KUKA KRL program: EPS_2_251806_MH43A_A_20260212042237.src

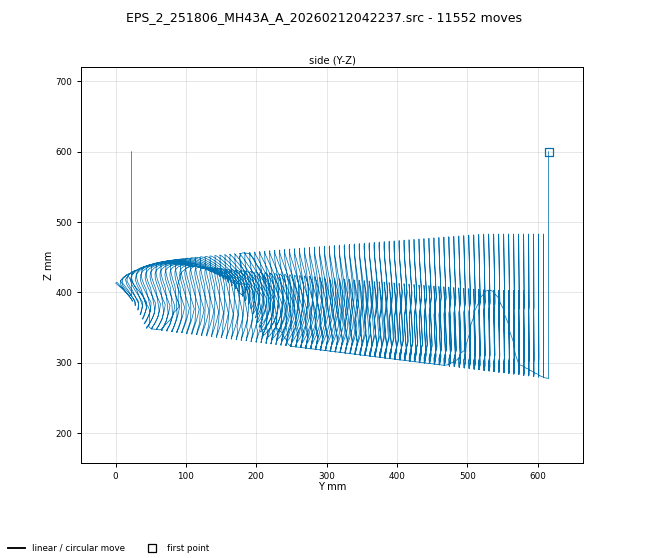
[picture p0: tool path of EPS_2_251806_MH43A_A_20260212042237.src, 11552 of 11554 moves have a stored position in this frame; points joined in program order, loops and branches not executed]
&ACCESS RVP
&REL 4
&COMMENT QRS 19112012
&PARAM EDITMASK = *
DEF PART()
EXT BAS (BAS_COMMAND :IN,REAL :IN )
INT I
BAS (#INITMOV,0 )

;KUKA QRS Post kuka4.cps  Date:22-06-2017 !

File_ID=3015

QRS_PRE_INIT()

;Init var - Until changes are made in qrs_pre_init
Outlet_Square_prg=0
Inlet_1_Square_prg=0
Inlet_2_Square_prg=0
Inlet_3_Square_prg=0
Inlet_4_Square_prg=0
Inlet_5_Square_prg=0

Outlet_1={X 0.000, Y 526.370, Z 382.500, B 0.000, E1 0.000 }
Inlet_1={X 0.000, Y 532.170, Z 302.500, B 0.000, E1 128.000 }
Outlet_1_type=201
Inlet_1_type=201
;QRS#1=Sidecore dimensions
;QRS#2=200-8" PVC SDR 35
;QRS#3=200-8" PVC SDR 35
;QRS#4=
;QRS#5=
;QRS#6=
;QRS#7=
;QRS#8=
;QRS#9=12-08 PSX
;QRS#10=12-08 PSX
;QRS#11=
;QRS#12=
;QRS#13=
;QRS#14=
;QRS#15=
;QRS#16=1220x127x762 2,5'
;QRS#17=EPS Height
;QRS#18=483
;QRS#19=*
;QRS#20= UPDATED VERSION 22-06-2017
;QRS#21=*
Outlet_Square=0100
Inlet_1_Square=0100
Inlet_2_Square=0
Inlet_3_Square=0
Inlet_4_Square=0
Inlet_5_Square=0
Mill_Square=1
Outlet_Square_Prg=204
Inlet_1_Square_prg=204

QRS_INIT()

$ADVANCE=5

; T1
PTP {E1 173.621,E2 173.621}
PTP {X 0,Y 615.489,A -85,B 0,C 180,E1 173.621,E2 173.621,E3 0,E4 0,E5 0,E6 0}
QRS_SPEED_INIT()
LIN {X 0,Y 615.489,Z 600,A -85,B 0,C 180,E1 173.621,E2 173.621,E3 0,E4 0,E5 0,E6 0} C_VEL
LIN {X 0,Y 615.489,Z 287.877,A -85,B 0,C 180,E1 173.621,E2 173.621} C_VEL
LIN {X 0,Y 615.489,Z 279.7,A -85,B 0,C 180,E1 173.621,E2 173.621} C_VEL
LIN {X 0,Y 615.478,Z 277.7,A -85,B 0,C 180,E1 173.435,E2 173.435} C_VEL
LIN {X 0,Y 615.494,Z 277.879,A -85,B 0,C 180,E1 170.801,E2 170.801} C_VEL
LIN {X 0,Y 615.483,Z 281.025,A -85,B 0,C 180,E1 168.139,E2 168.139} C_VEL
LIN {X 0,Y 615.467,Z 284.295,A -85,B 0,C 180,E1 165.451,E2 165.451} C_VEL
LIN {X 0,Y 615.488,Z 287.642,A -85,B 0,C 180,E1 162.73,E2 162.73} C_VEL
LIN {X 0,Y 615.467,Z 291.126,A -85,B 0,C 180,E1 159.967,E2 159.967} C_VEL
LIN {X 0,Y 615.473,Z 294.079,A -85,B 0,C 180,E1 157.659,E2 157.659} C_VEL
LIN {X 0,Y 615.485,Z 297.487,A -85,B 0,C 180,E1 155.008,E2 155.008} C_VEL
LIN {X 0,Y 615.484,Z 299.412,A -85,B 0,C 180,E1 153.537,E2 153.537} C_VEL
LIN {X 0,Y 615.487,Z 313.298,A -85,B 0,C 180,E1 153.219,E2 153.219} C_VEL
LIN {X 0,Y 615.486,Z 325.134,A -85,B 0,C 180,E1 152.823,E2 152.823} C_VEL
LIN {X 0,Y 615.476,Z 337.354,A -85,B 0,C 180,E1 152.269,E2 152.269} C_VEL
LIN {X 0,Y 615.49,Z 348.526,A -85,B 0,C 180,E1 151.617,E2 151.617} C_VEL
LIN {X 0,Y 615.5,Z 358.718,A -85,B 0,C 180,E1 150.876,E2 150.876} C_VEL
LIN {X 0,Y 615.498,Z 368.21,A -85,B 0,C 180,E1 150.023,E2 150.023} C_VEL
LIN {X 0,Y 615.497,Z 376.7,A -85,B 0,C 180,E1 149.081,E2 149.081} C_VEL
LIN {X 0,Y 615.498,Z 383.506,A -85,B 0,C 180,E1 148.154,E2 148.154} C_VEL
LIN {X 0,Y 615.495,Z 389.434,A -85,B 0,C 180,E1 147.154,E2 147.154} C_VEL
LIN {X 0,Y 615.495,Z 394.786,A -85,B 0,C 180,E1 145.979,E2 145.979} C_VEL
LIN {X 0,Y 615.497,Z 398.663,A -85,B 0,C 180,E1 144.786,E2 144.786} C_VEL
LIN {X 0,Y 615.494,Z 401.179,A -85,B 0,C 180,E1 143.576,E2 143.576} C_VEL
LIN {X 0,Y 615.496,Z 402.068,A -85,B 0,C 180,E1 142.758,E2 142.758} C_VEL
LIN {X 0,Y 615.494,Z 402.388,A -85,B 0,C 180,E1 141.932,E2 141.932} C_VEL
LIN {X 0,Y 615.495,Z 401.915,A -85,B 0,C 180,E1 140.938,E2 140.938} C_VEL
LIN {X 0,Y 615.496,Z 400.472,A -85,B 0,C 180,E1 139.911,E2 139.911} C_VEL
LIN {X 0,Y 615.494,Z 398.079,A -85,B 0,C 180,E1 138.905,E2 138.905} C_VEL
LIN {X 0,Y 615.497,Z 394.741,A -85,B 0,C 180,E1 137.92,E2 137.92} C_VEL
LIN {X 0,Y 615.498,Z 389.437,A -85,B 0,C 180,E1 136.756,E2 136.756} C_VEL
LIN {X 0,Y 615.494,Z 382.833,A -85,B 0,C 180,E1 135.656,E2 135.656} C_VEL
LIN {X 0,Y 615.495,Z 375.934,A -85,B 0,C 180,E1 134.736,E2 134.736} C_VEL
LIN {X 0,Y 615.498,Z 367.434,A -85,B 0,C 180,E1 133.809,E2 133.809} C_VEL
LIN {X 0,Y 615.499,Z 357.779,A -85,B 0,C 180,E1 132.961,E2 132.961} C_VEL
LIN {X 0,Y 615.481,Z 347.336,A -85,B 0,C 180,E1 132.216,E2 132.216} C_VEL
LIN {X 0,Y 615.461,Z 337.097,A -85,B 0,C 180,E1 131.627,E2 131.627} C_VEL
LIN {X 0,Y 615.487,Z 325.327,A -85,B 0,C 180,E1 131.094,E2 131.094} C_VEL
LIN {X 0,Y 615.492,Z 312.445,A -85,B 0,C 180,E1 130.667,E2 130.667} C_VEL
LIN {X 0,Y 615.482,Z 299.399,A -85,B 0,C 180,E1 130.362,E2 130.362} C_VEL
LIN {X 0,Y 615.455,Z 296.342,A -85,B 0,C 180,E1 128.008,E2 128.008} C_VEL
LIN {X 0,Y 615.46,Z 293.257,A -85,B 0,C 180,E1 125.618,E2 125.618} C_VEL
LIN {X 0,Y 615.488,Z 290.222,A -85,B 0,C 180,E1 123.237,E2 123.237} C_VEL
LIN {X 0,Y 615.496,Z 287.32,A -85,B 0,C 180,E1 120.92,E2 120.92} C_VEL
LIN {X 0,Y 615.458,Z 284.279,A -85,B 0,C 180,E1 118.445,E2 118.445} C_VEL
LIN {X 0,Y 615.454,Z 281.851,A -85,B 0,C 180,E1 116.446,E2 116.446} C_VEL
LIN {X 0,Y 615.451,Z 278.929,A -85,B 0,C 180,E1 114.001,E2 114.001} C_VEL
LIN {X 0,Y 615.477,Z 277.7,A -85,B 0,C 180,E1 112.845,E2 112.845} C_VEL
LIN {X 0,Y 615.481,Z 277.697,A -85,B 0,C 180,E1 110.033,E2 110.033} C_VEL
LIN {X 0,Y 615.476,Z 277.697,A -85,B 0,C 180,E1 107.271,E2 107.271} C_VEL
LIN {X 0,Y 615.46,Z 277.7,A -85,B 0,C 180,E1 104.55,E2 104.55} C_VEL
LIN {X 0,Y 615.487,Z 277.694,A -85,B 0,C 180,E1 101.861,E2 101.861} C_VEL
LIN {X 0,Y 615.468,Z 277.698,A -85,B 0,C 180,E1 99.199,E2 99.199} C_VEL
LIN {X 0,Y 615.461,Z 277.7,A -85,B 0,C 180,E1 96.556,E2 96.556} C_VEL
LIN {X 0,Y 615.491,Z 277.693,A -85,B 0,C 180,E1 93.929,E2 93.929} C_VEL
LIN {X 0,Y 615.466,Z 277.699,A -85,B 0,C 180,E1 91.309,E2 91.309} C_VEL
LIN {X 0,Y 615.461,Z 277.7,A -85,B 0,C 180,E1 88.691,E2 88.691} C_VEL
LIN {X 0,Y 615.491,Z 277.693,A -85,B 0,C 180,E1 86.071,E2 86.071} C_VEL
LIN {X 0,Y 615.465,Z 277.699,A -85,B 0,C 180,E1 83.441,E2 83.441} C_VEL
LIN {X 0,Y 615.461,Z 277.7,A -85,B 0,C 180,E1 80.801,E2 80.801} C_VEL
LIN {X 0,Y 615.49,Z 277.694,A -85,B 0,C 180,E1 78.139,E2 78.139} C_VEL
LIN {X 0,Y 615.465,Z 277.7,A -85,B 0,C 180,E1 75.45,E2 75.45} C_VEL
LIN {X 0,Y 615.47,Z 277.7,A -85,B 0,C 180,E1 72.729,E2 72.729} C_VEL
LIN {X 0,Y 615.49,Z 277.697,A -85,B 0,C 180,E1 69.967,E2 69.967} C_VEL
LIN {X 0,Y 615.487,Z 277.703,A -85,B 0,C 180,E1 67.155,E2 67.155} C_VEL
LIN {X 0,Y 615.477,Z 277.7,A -85,B 0,C 180,E1 64.284,E2 64.284} C_VEL
LIN {X 0,Y 615.469,Z 277.7,A -85,B 0,C 180,E1 61.553,E2 61.553} C_VEL
LIN {X 0,Y 615.493,Z 277.695,A -85,B 0,C 180,E1 58.913,E2 58.913} C_VEL
LIN {X 0,Y 615.459,Z 277.7,A -85,B 0,C 180,E1 55.976,E2 55.976} C_VEL
LIN {X 0,Y 615.47,Z 277.699,A -85,B 0,C 180,E1 53.574,E2 53.574} C_VEL
LIN {X 0,Y 615.497,Z 277.692,A -85,B 0,C 180,E1 50.937,E2 50.937} C_VEL
LIN {X 0,Y 615.477,Z 277.7,A -85,B 0,C 180,E1 48.525,E2 48.525} C_VEL
LIN {X 0,Y 615.477,Z 277.699,A -85,B 0,C 180,E1 45.849,E2 45.849} C_VEL
LIN {X 0,Y 615.491,Z 277.694,A -85,B 0,C 180,E1 43.047,E2 43.047} C_VEL
LIN {X 0,Y 615.47,Z 277.701,A -85,B 0,C 180,E1 40.608,E2 40.608} C_VEL
LIN {X 0,Y 615.48,Z 277.699,A -85,B 0,C 180,E1 38.01,E2 38.01} C_VEL
LIN {X 0,Y 615.499,Z 277.7,A -85,B 0,C 180,E1 35.615,E2 35.615} C_VEL
LIN {X 0,Y 615.491,Z 277.697,A -85,B 0,C 180,E1 33.236,E2 33.236} C_VEL
LIN {X 0,Y 615.481,Z 277.696,A -85,B 0,C 180,E1 30.92,E2 30.92} C_VEL
LIN {X 0,Y 615.459,Z 277.7,A -85,B 0,C 180,E1 28.444,E2 28.444} C_VEL
LIN {X 0,Y 615.477,Z 277.696,A -85,B 0,C 180,E1 25.716,E2 25.716} C_VEL
LIN {X 0,Y 615.48,Z 277.698,A -85,B 0,C 180,E1 22.845,E2 22.845} C_VEL
LIN {X 0,Y 615.46,Z 277.7,A -85,B 0,C 180,E1 20.549,E2 20.549} C_VEL
LIN {X 0,Y 615.48,Z 277.696,A -85,B 0,C 180,E1 17.957,E2 17.957} C_VEL
LIN {X 0,Y 615.477,Z 277.696,A -85,B 0,C 180,E1 15.226,E2 15.226} C_VEL
LIN {X 0,Y 615.46,Z 277.7,A -85,B 0,C 180,E1 12.531,E2 12.531} C_VEL
LIN {X 0,Y 615.494,Z 277.693,A -85,B 0,C 180,E1 9.862,E2 9.862} C_VEL
LIN {X 0,Y 615.474,Z 277.698,A -85,B 0,C 180,E1 7.216,E2 7.216} C_VEL
LIN {X 0,Y 615.463,Z 277.7,A -85,B 0,C 180,E1 4.585,E2 4.585} C_VEL
LIN {X 0,Y 615.5,Z 277.692,A -85,B 0,C 180,E1 1.963,E2 1.963} C_VEL
LIN {X 0,Y 615.472,Z 277.698,A -85,B 0,C 180,E1 -0.654,E2 -0.654} C_VEL
LIN {X 0,Y 615.461,Z 277.701,A -85,B 0,C 180,E1 -3.273,E2 -3.273} C_VEL
LIN {X 0,Y 615.499,Z 277.692,A -85,B 0,C 180,E1 -5.899,E2 -5.899} C_VEL
LIN {X 0,Y 615.47,Z 277.699,A -85,B 0,C 180,E1 -8.537,E2 -8.537} C_VEL
LIN {X 0,Y 615.463,Z 277.7,A -85,B 0,C 180,E1 -11.194,E2 -11.194} C_VEL
LIN {X 0,Y 615.493,Z 277.695,A -85,B 0,C 180,E1 -13.933,E2 -13.933} C_VEL
LIN {X 0,Y 615.476,Z 277.699,A -85,B 0,C 180,E1 -16.587,E2 -16.587} C_VEL
LIN {X 0,Y 615.481,Z 277.701,A -85,B 0,C 180,E1 -19.338,E2 -19.338} C_VEL
LIN {X 0,Y 615.494,Z 277.701,A -85,B 0,C 180,E1 -22.136,E2 -22.136} C_VEL
LIN {X 0,Y 615.488,Z 277.697,A -85,B 0,C 180,E1 -24.992,E2 -24.992} C_VEL
LIN {X 0,Y 615.463,Z 277.7,A -85,B 0,C 180,E1 -27.916,E2 -27.916} C_VEL
LIN {X 0,Y 615.482,Z 277.7,A -85,B 0,C 180,E1 -30.161,E2 -30.161} C_VEL
LIN {X 0,Y 615.481,Z 277.7,A -85,B 0,C 180,E1 -32.458,E2 -32.458} C_VEL
LIN {X 0,Y 615.467,Z 277.7,A -85,B 0,C 180,E1 -34.817,E2 -34.817} C_VEL
LIN {X 0,Y 615.495,Z 277.692,A -85,B 0,C 180,E1 -37.242,E2 -37.242} C_VEL
LIN {X 0,Y 615.463,Z 277.701,A -85,B 0,C 180,E1 -40.086,E2 -40.086} C_VEL
LIN {X 0,Y 615.465,Z 277.699,A -85,B 0,C 180,E1 -42.355,E2 -42.355} C_VEL
LIN {X 0,Y 615.493,Z 277.693,A -85,B 0,C 180,E1 -45.068,E2 -45.068} C_VEL
LIN {X 0,Y 615.464,Z 277.7,A -85,B 0,C 180,E1 -47.923,E2 -47.923} C_VEL
LIN {X 0,Y 615.466,Z 277.699,A -85,B 0,C 180,E1 -50.248,E2 -50.248} C_VEL
LIN {X 0,Y 615.488,Z 277.694,A -85,B 0,C 180,E1 -53.064,E2 -53.064} C_VEL
LIN {X 0,Y 615.479,Z 277.84,A -85,B 0,C 180,E1 -54.584,E2 -54.584} C_VEL
LIN {X 0,Y 615.491,Z 287.498,A -85,B 0,C 180,E1 -57.154,E2 -57.154} C_VEL
LIN {X 0,Y 615.485,Z 297.895,A -85,B 0,C 180,E1 -59.839,E2 -59.839} C_VEL
LIN {X 0,Y 615.485,Z 308.132,A -85,B 0,C 180,E1 -62.454,E2 -62.454} C_VEL
LIN {X 0,Y 615.444,Z 319.822,A -85,B 0,C 180,E1 -65.367,E2 -65.367} C_VEL
LIN {X 0,Y 615.447,Z 330.043,A -85,B 0,C 180,E1 -67.862,E2 -67.862} C_VEL
LIN {X 0,Y 615.477,Z 341.714,A -85,B 0,C 180,E1 -70.662,E2 -70.662} C_VEL
LIN {X 0,Y 615.485,Z 353.374,A -85,B 0,C 180,E1 -73.413,E2 -73.413} C_VEL
LIN {X 0,Y 615.485,Z 365.04,A -85,B 0,C 180,E1 -76.126,E2 -76.126} C_VEL
LIN {X 0,Y 615.497,Z 374.676,A -85,B 0,C 180,E1 -78.348,E2 -78.348} C_VEL
LIN {X 0,Y 615.496,Z 388.059,A -85,B 0,C 180,E1 -78.598,E2 -78.598} C_VEL
LIN {X 0,Y 615.471,Z 400.703,A -85,B 0,C 180,E1 -78.967,E2 -78.967} C_VEL
LIN {X 0,Y 615.447,Z 413.027,A -85,B 0,C 180,E1 -79.472,E2 -79.472} C_VEL
LIN {X 0,Y 615.48,Z 423.981,A -85,B 0,C 180,E1 -80.055,E2 -80.055} C_VEL
LIN {X 0,Y 615.499,Z 435.166,A -85,B 0,C 180,E1 -80.801,E2 -80.801} C_VEL
LIN {X 0,Y 615.498,Z 445.044,A -85,B 0,C 180,E1 -81.629,E2 -81.629} C_VEL
LIN {X 0,Y 615.498,Z 454.606,A -85,B 0,C 180,E1 -82.62,E2 -82.62} C_VEL
LIN {X 0,Y 615.496,Z 462.203,A -85,B 0,C 180,E1 -83.608,E2 -83.608} C_VEL
LIN {X 0,Y 615.498,Z 469.204,A -85,B 0,C 180,E1 -84.759,E2 -84.759} C_VEL
LIN {X 0,Y 615.494,Z 473.851,A -85,B 0,C 180,E1 -85.744,E2 -85.744} C_VEL
LIN {X 0,Y 615.494,Z 477.399,A -85,B 0,C 180,E1 -86.727,E2 -86.727} C_VEL
LIN {X 0,Y 615.497,Z 479.233,A -85,B 0,C 180,E1 -87.382,E2 -87.382} C_VEL
LIN {X 0,Y 615.5,Z 480.607,A -85,B 0,C 180,E1 -88.037,E2 -88.037} C_VEL
LIN {X 0,Y 615.496,Z 482.173,A -85,B 0,C 180,E1 -89.346,E2 -89.346} C_VEL
LIN {X 0,Y 615.494,Z 482.389,A -85,B 0,C 180,E1 -90,E2 -90} C_VEL
LIN {X 0,Y 615.495,Z 481.58,A -85,B 0,C 180,E1 -91.309,E2 -91.309} C_VEL
LIN {X 0,Y 615.5,Z 480.607,A -85,B 0,C 180,E1 -91.963,E2 -91.963} C_VEL
LIN {X 0,Y 615.497,Z 479.233,A -85,B 0,C 180,E1 -92.618,E2 -92.618} C_VEL
LIN {X 0,Y 615.496,Z 476.349,A -85,B 0,C 180,E1 -93.601,E2 -93.601} C_VEL
LIN {X 0,Y 615.498,Z 472.441,A -85,B 0,C 180,E1 -94.585,E2 -94.585} C_VEL
LIN {X 0,Y 615.499,Z 467.404,A -85,B 0,C 180,E1 -95.57,E2 -95.57} C_VEL
LIN {X 0,Y 615.497,Z 460.87,A -85,B 0,C 180,E1 -96.583,E2 -96.583} C_VEL
LIN {X 0,Y 615.497,Z 453.132,A -85,B 0,C 180,E1 -97.545,E2 -97.545} C_VEL
LIN {X 0,Y 615.498,Z 445.044,A -85,B 0,C 180,E1 -98.371,E2 -98.371} C_VEL
LIN {X 0,Y 615.499,Z 435.166,A -85,B 0,C 180,E1 -99.199,E2 -99.199} C_VEL
LIN {X 0,Y 615.48,Z 423.981,A -85,B 0,C 180,E1 -99.945,E2 -99.945} C_VEL
LIN {X 0,Y 615.447,Z 413.027,A -85,B 0,C 180,E1 -100.528,E2 -100.528} C_VEL
LIN {X 0,Y 615.471,Z 400.703,A -85,B 0,C 180,E1 -101.033,E2 -101.033} C_VEL
LIN {X 0,Y 615.496,Z 388.058,A -85,B 0,C 180,E1 -101.402,E2 -101.402} C_VEL
LIN {X 0,Y 615.497,Z 374.676,A -85,B 0,C 180,E1 -101.652,E2 -101.652} C_VEL
LIN {X 0,Y 615.48,Z 362.118,A -85,B 0,C 180,E1 -104.549,E2 -104.549} C_VEL
LIN {X 0,Y 615.475,Z 350.467,A -85,B 0,C 180,E1 -107.271,E2 -107.271} C_VEL
LIN {X 0,Y 615.483,Z 338.793,A -85,B 0,C 180,E1 -110.033,E2 -110.033} C_VEL
LIN {X 0,Y 615.43,Z 328.185,A -85,B 0,C 180,E1 -112.59,E2 -112.59} C_VEL
LIN {X 0,Y 615.492,Z 317.195,A -85,B 0,C 180,E1 -115.279,E2 -115.279} C_VEL
LIN {X 0,Y 615.466,Z 306.67,A -85,B 0,C 180,E1 -117.916,E2 -117.916} C_VEL
LIN {X 0,Y 615.487,Z 296.432,A -85,B 0,C 180,E1 -120.539,E2 -120.539} C_VEL
LIN {X 0,Y 615.492,Z 285.882,A -85,B 0,C 180,E1 -123.236,E2 -123.236} C_VEL
LIN {X 0,Y 615.483,Z 277.699,A -85,B 0,C 180,E1 -125.416,E2 -125.416} C_VEL
LIN {X 0,Y 615.487,Z 277.702,A -85,B 0,C 180,E1 -128.069,E2 -128.069} C_VEL
LIN {X 0,Y 615.477,Z 277.7,A -85,B 0,C 180,E1 -130.608,E2 -130.608} C_VEL
LIN {X 0,Y 615.485,Z 277.7,A -85,B 0,C 180,E1 -133.245,E2 -133.245} C_VEL
LIN {X 0,Y 615.486,Z 277.702,A -85,B 0,C 180,E1 -136.003,E2 -136.003} C_VEL
LIN {X 0,Y 615.492,Z 277.699,A -85,B 0,C 180,E1 -138.906,E2 -138.906} C_VEL
LIN {X 0,Y 615.496,Z 277.7,A -85,B 0,C 180,E1 -141.096,E2 -141.096} C_VEL
LIN {X 0,Y 615.475,Z 277.7,A -85,B 0,C 180,E1 -143.574,E2 -143.574} C_VEL
LIN {X 0,Y 615.49,Z 277.697,A -85,B 0,C 180,E1 -146.466,E2 -146.466} C_VEL
LIN {X 0,Y 615.493,Z 277.702,A -85,B 0,C 180,E1 -149.08,E2 -149.08} C_VEL
LIN {X 0,Y 615.477,Z 277.7,A -85,B 0,C 180,E1 -151.553,E2 -151.553} C_VEL
LIN {X 0,Y 615.495,Z 277.698,A -85,B 0,C 180,E1 -154.284,E2 -154.284} C_VEL
LIN {X 0,Y 615.487,Z 277.702,A -85,B 0,C 180,E1 -157.155,E2 -157.155} C_VEL
LIN {X 0,Y 615.483,Z 277.701,A -85,B 0,C 180,E1 -159.967,E2 -159.967} C_VEL
LIN {X 0,Y 615.488,Z 277.698,A -85,B 0,C 180,E1 -162.729,E2 -162.729} C_VEL
LIN {X 0,Y 615.478,Z 277.7,A -85,B 0,C 180,E1 -165.451,E2 -165.451} C_VEL
LIN {X 0,Y 615.491,Z 277.702,A -85,B 0,C 180,E1 -168.139,E2 -168.139} C_VEL
LIN {X 0,Y 615.481,Z 277.7,A -85,B 0,C 180,E1 -170.801,E2 -170.801} C_VEL
LIN {X 0,Y 615.48,Z 277.7,A -85,B 0,C 180,E1 -173.443,E2 -173.443} C_VEL
LIN {X 0,Y 615.488,Z 277.701,A -85,B 0,C 180,E1 -176.071,E2 -176.071} C_VEL
LIN {X 0,Y 615.477,Z 277.7,A -85,B 0,C 180,E1 -178.691,E2 -178.691} C_VEL
LIN {X 0,Y 615.488,Z 277.7,A -85,B 0,C 180,E1 -181.309,E2 -181.309} C_VEL
LIN {X 0,Y 615.493,Z 277.698,A -85,B 0,C 180,E1 -183.928,E2 -183.928} C_VEL
LIN {X 0,Y 615.478,Z 277.7,A -85,B 0,C 180,E1 -186.565,E2 -186.565} C_VEL
LIN {X 0,Y 614.804,Z 277.846,A -85,B 0,C 180,E1 -187.112,E2 -187.112} C_VEL
LIN {X 0,Y 611.956,Z 278.261,A -85,B 0,C 180,E1 -187.999,E2 -187.999} C_VEL
LIN {X 0,Y 609.551,Z 278.559,A -85,B 0,C 180,E1 -188.711,E2 -188.711} C_VEL
LIN {X 0,Y 608.51,Z 278.76,A -85,B 0,C 180,E1 -189.26,E2 -189.26} C_VEL
LIN {X 0,Y 608.421,Z 278.929,A -85,B 0,C 180,E1 -189.445,E2 -189.445} C_VEL
LIN {X 0,Y 608.418,Z 281.945,A -85,B 0,C 180,E1 -192.001,E2 -192.001} C_VEL
LIN {X 0,Y 608.405,Z 285.23,A -85,B 0,C 180,E1 -194.722,E2 -194.722} C_VEL
LIN {X 0,Y 608.411,Z 287.765,A -85,B 0,C 180,E1 -196.785,E2 -196.785} C_VEL
LIN {X 0,Y 608.407,Z 291.246,A -85,B 0,C 180,E1 -199.572,E2 -199.572} C_VEL
LIN {X 0,Y 608.434,Z 294.925,A -85,B 0,C 180,E1 -202.469,E2 -202.469} C_VEL
LIN {X 0,Y 608.431,Z 298.573,A -85,B 0,C 180,E1 -205.302,E2 -205.302} C_VEL
LIN {X 0,Y 608.409,Z 299.917,A -85,B 0,C 180,E1 -206.337,E2 -206.337} C_VEL
LIN {X 0,Y 608.547,Z 313.537,A -85,B 0,C 180,E1 -206.654,E2 -206.654} C_VEL
LIN {X 0,Y 608.533,Z 325.841,A -85,B 0,C 180,E1 -207.074,E2 -207.074} C_VEL
LIN {X 0,Y 608.48,Z 337.496,A -85,B 0,C 180,E1 -207.61,E2 -207.61} C_VEL
LIN {X 0,Y 608.475,Z 348.646,A -85,B 0,C 180,E1 -208.265,E2 -208.265} C_VEL
LIN {X 0,Y 608.493,Z 358.943,A -85,B 0,C 180,E1 -209.019,E2 -209.019} C_VEL
LIN {X 0,Y 608.483,Z 367.48,A -85,B 0,C 180,E1 -209.779,E2 -209.779} C_VEL
LIN {X 0,Y 608.459,Z 376.169,A -85,B 0,C 180,E1 -210.726,E2 -210.726} C_VEL
LIN {X 0,Y 608.464,Z 383.466,A -85,B 0,C 180,E1 -211.705,E2 -211.705} C_VEL
LIN {X 0,Y 608.432,Z 388.449,A -85,B 0,C 180,E1 -212.517,E2 -212.517} C_VEL
LIN {X 0,Y 608.425,Z 394.321,A -85,B 0,C 180,E1 -213.727,E2 -213.727} C_VEL
LIN {X 0,Y 608.427,Z 398.483,A -85,B 0,C 180,E1 -214.902,E2 -214.902} C_VEL
LIN {X 0,Y 608.424,Z 401.259,A -85,B 0,C 180,E1 -216.094,E2 -216.094} C_VEL
LIN {X 0,Y 608.435,Z 402.622,A -85,B 0,C 180,E1 -217.153,E2 -217.153} C_VEL
LIN {X 0,Y 608.421,Z 402.962,A -85,B 0,C 180,E1 -218.234,E2 -218.234} C_VEL
LIN {X 0,Y 608.424,Z 402.096,A -85,B 0,C 180,E1 -219.443,E2 -219.443} C_VEL
LIN {X 0,Y 608.434,Z 399.687,A -85,B 0,C 180,E1 -220.74,E2 -220.74} C_VEL
LIN {X 0,Y 608.45,Z 396.944,A -85,B 0,C 180,E1 -221.673,E2 -221.673} C_VEL
LIN {X 0,Y 608.442,Z 393.222,A -85,B 0,C 180,E1 -222.619,E2 -222.619} C_VEL
LIN {X 0,Y 608.453,Z 388.512,A -85,B 0,C 180,E1 -223.561,E2 -223.561} C_VEL
LIN {X 0,Y 608.46,Z 381.686,A -85,B 0,C 180,E1 -224.648,E2 -224.648} C_VEL
LIN {X 0,Y 608.469,Z 372.971,A -85,B 0,C 180,E1 -225.735,E2 -225.735} C_VEL
LIN {X 0,Y 608.476,Z 364.475,A -85,B 0,C 180,E1 -226.595,E2 -226.595} C_VEL
LIN {X 0,Y 608.48,Z 354.949,A -85,B 0,C 180,E1 -227.384,E2 -227.384} C_VEL
LIN {X 0,Y 608.477,Z 343.675,A -85,B 0,C 180,E1 -228.135,E2 -228.135} C_VEL
LIN {X 0,Y 608.5,Z 331.524,A -85,B 0,C 180,E1 -228.773,E2 -228.773} C_VEL
LIN {X 0,Y 608.537,Z 318.931,A -85,B 0,C 180,E1 -229.268,E2 -229.268} C_VEL
LIN {X 0,Y 608.555,Z 305.75,A -85,B 0,C 180,E1 -229.634,E2 -229.634} C_VEL
LIN {X 0,Y 608.418,Z 299.903,A -85,B 0,C 180,E1 -229.764,E2 -229.764} C_VEL
LIN {X 0,Y 608.431,Z 295.917,A -85,B 0,C 180,E1 -232.846,E2 -232.846} C_VEL
LIN {X 0,Y 608.405,Z 292.499,A -85,B 0,C 180,E1 -235.526,E2 -235.526} C_VEL
LIN {X 0,Y 608.388,Z 289.512,A -85,B 0,C 180,E1 -237.901,E2 -237.901} C_VEL
LIN {X 0,Y 608.409,Z 286.639,A -85,B 0,C 180,E1 -240.217,E2 -240.217} C_VEL
LIN {X 0,Y 608.435,Z 283.49,A -85,B 0,C 180,E1 -242.801,E2 -242.801} C_VEL
LIN {X 0,Y 608.406,Z 280.359,A -85,B 0,C 180,E1 -245.427,E2 -245.427} C_VEL
LIN {X 0,Y 608.418,Z 278.703,A -85,B 0,C 180,E1 -246.874,E2 -246.874} C_VEL
LIN {X 0,Y 608.469,Z 278.694,A -85,B 0,C 180,E1 -249.321,E2 -249.321} C_VEL
LIN {X 0,Y 608.44,Z 278.696,A -85,B 0,C 180,E1 -251.828,E2 -251.828} C_VEL
LIN {X 0,Y 608.475,Z 278.693,A -85,B 0,C 180,E1 -254.594,E2 -254.594} C_VEL
LIN {X 0,Y 608.475,Z 278.694,A -85,B 0,C 180,E1 -257.323,E2 -257.323} C_VEL
LIN {X 0,Y 608.461,Z 278.697,A -85,B 0,C 180,E1 -260.023,E2 -260.023} C_VEL
LIN {X 0,Y 608.462,Z 278.697,A -85,B 0,C 180,E1 -262.701,E2 -262.701} C_VEL
LIN {X 0,Y 608.459,Z 278.697,A -85,B 0,C 180,E1 -265.362,E2 -265.362} C_VEL
LIN {X 0,Y 608.468,Z 278.695,A -85,B 0,C 180,E1 -268.014,E2 -268.014} C_VEL
LIN {X 0,Y 608.477,Z 278.694,A -85,B 0,C 180,E1 -270.662,E2 -270.662} C_VEL
LIN {X 0,Y 608.486,Z 278.692,A -85,B 0,C 180,E1 -273.311,E2 -273.311} C_VEL
LIN {X 0,Y 608.467,Z 278.695,A -85,B 0,C 180,E1 -275.967,E2 -275.967} C_VEL
LIN {X 0,Y 608.45,Z 278.696,A -85,B 0,C 180,E1 -278.636,E2 -278.636} C_VEL
LIN {X 0,Y 608.482,Z 278.692,A -85,B 0,C 180,E1 -281.324,E2 -281.324} C_VEL
LIN {X 0,Y 608.448,Z 278.695,A -85,B 0,C 180,E1 -284.038,E2 -284.038} C_VEL
LIN {X 0,Y 608.474,Z 278.693,A -85,B 0,C 180,E1 -286.531,E2 -286.531} C_VEL
LIN {X 0,Y 608.455,Z 278.693,A -85,B 0,C 180,E1 -289.571,E2 -289.571} C_VEL
LIN {X 0,Y 608.461,Z 278.693,A -85,B 0,C 180,E1 -292.477,E2 -292.477} C_VEL
LIN {X 0,Y 608.446,Z 278.695,A -85,B 0,C 180,E1 -294.572,E2 -294.572} C_VEL
LIN {X 0,Y 608.485,Z 278.69,A -85,B 0,C 180,E1 -297.208,E2 -297.208} C_VEL
LIN {X 0,Y 608.432,Z 278.696,A -85,B 0,C 180,E1 -299.966,E2 -299.966} C_VEL
LIN {X 0,Y 608.448,Z 278.694,A -85,B 0,C 180,E1 -302.52,E2 -302.52} C_VEL
LIN {X 0,Y 608.445,Z 278.694,A -85,B 0,C 180,E1 -305.278,E2 -305.278} C_VEL
LIN {X 0,Y 608.455,Z 278.694,A -85,B 0,C 180,E1 -307.748,E2 -307.748} C_VEL
LIN {X 0,Y 608.443,Z 278.695,A -85,B 0,C 180,E1 -310.328,E2 -310.328} C_VEL
LIN {X 0,Y 608.476,Z 278.691,A -85,B 0,C 180,E1 -313.309,E2 -313.309} C_VEL
LIN {X 0,Y 608.454,Z 278.694,A -85,B 0,C 180,E1 -316.129,E2 -316.129} C_VEL
LIN {X 0,Y 608.455,Z 278.695,A -85,B 0,C 180,E1 -318.823,E2 -318.823} C_VEL
LIN {X 0,Y 608.47,Z 278.693,A -85,B 0,C 180,E1 -321.412,E2 -321.412} C_VEL
LIN {X 0,Y 608.445,Z 278.695,A -85,B 0,C 180,E1 -323.955,E2 -323.955} C_VEL
LIN {X 0,Y 608.446,Z 278.694,A -85,B 0,C 180,E1 -326.328,E2 -326.328} C_VEL
LIN {X 0,Y 608.451,Z 278.694,A -85,B 0,C 180,E1 -328.733,E2 -328.733} C_VEL
LIN {X 0,Y 608.454,Z 278.694,A -85,B 0,C 180,E1 -331.384,E2 -331.384} C_VEL
LIN {X 0,Y 608.442,Z 278.695,A -85,B 0,C 180,E1 -333.964,E2 -333.964} C_VEL
LIN {X 0,Y 608.451,Z 278.694,A -85,B 0,C 180,E1 -336.876,E2 -336.876} C_VEL
LIN {X 0,Y 608.449,Z 278.694,A -85,B 0,C 180,E1 -339.327,E2 -339.327} C_VEL
LIN {X 0,Y 608.447,Z 278.695,A -85,B 0,C 180,E1 -341.828,E2 -341.828} C_VEL
LIN {X 0,Y 608.467,Z 278.692,A -85,B 0,C 180,E1 -344.594,E2 -344.594} C_VEL
LIN {X 0,Y 608.458,Z 278.693,A -85,B 0,C 180,E1 -347.323,E2 -347.323} C_VEL
LIN {X 0,Y 608.463,Z 278.692,A -85,B 0,C 180,E1 -350.023,E2 -350.023} C_VEL
LIN {X 0,Y 608.444,Z 278.695,A -85,B 0,C 180,E1 -352.7,E2 -352.7} C_VEL
LIN {X 0,Y 608.432,Z 278.696,A -85,B 0,C 180,E1 -355.362,E2 -355.362} C_VEL
LIN {X 0,Y 608.469,Z 278.692,A -85,B 0,C 180,E1 -358.014,E2 -358.014} C_VEL
LIN {X 0,Y 608.469,Z 278.692,A -85,B 0,C 180,E1 -360.662,E2 -360.662} C_VEL
LIN {X 0,Y 608.431,Z 278.697,A -85,B 0,C 180,E1 -363.311,E2 -363.311} C_VEL
LIN {X 0,Y 608.47,Z 278.692,A -85,B 0,C 180,E1 -365.967,E2 -365.967} C_VEL
LIN {X 0,Y 608.445,Z 278.695,A -85,B 0,C 180,E1 -368.636,E2 -368.636} C_VEL
LIN {X 0,Y 608.436,Z 278.697,A -85,B 0,C 180,E1 -371.325,E2 -371.325} C_VEL
LIN {X 0,Y 608.476,Z 278.693,A -85,B 0,C 180,E1 -374.037,E2 -374.037} C_VEL
LIN {X 0,Y 608.443,Z 278.699,A -85,B 0,C 180,E1 -376.784,E2 -376.784} C_VEL
LIN {X 0,Y 608.442,Z 278.699,A -85,B 0,C 180,E1 -379.571,E2 -379.571} C_VEL
LIN {X 0,Y 608.477,Z 278.691,A -85,B 0,C 180,E1 -381.691,E2 -381.691} C_VEL
LIN {X 0,Y 608.445,Z 278.697,A -85,B 0,C 180,E1 -384.572,E2 -384.572} C_VEL
LIN {X 0,Y 608.47,Z 278.694,A -85,B 0,C 180,E1 -387.205,E2 -387.205} C_VEL
LIN {X 0,Y 608.47,Z 278.696,A -85,B 0,C 180,E1 -389.971,E2 -389.971} C_VEL
LIN {X 0,Y 608.459,Z 278.694,A -85,B 0,C 180,E1 -392.88,E2 -392.88} C_VEL
LIN {X 0,Y 608.427,Z 278.701,A -85,B 0,C 180,E1 -395.279,E2 -395.279} C_VEL
LIN {X 0,Y 608.469,Z 278.695,A -85,B 0,C 180,E1 -397.746,E2 -397.746} C_VEL
LIN {X 0,Y 608.443,Z 278.698,A -85,B 0,C 180,E1 -400.327,E2 -400.327} C_VEL
LIN {X 0,Y 608.474,Z 278.693,A -85,B 0,C 180,E1 -403.309,E2 -403.309} C_VEL
LIN {X 0,Y 608.463,Z 278.693,A -85,B 0,C 180,E1 -406.13,E2 -406.13} C_VEL
LIN {X 0,Y 608.46,Z 278.693,A -85,B 0,C 180,E1 -408.823,E2 -408.823} C_VEL
LIN {X 0,Y 608.455,Z 278.693,A -85,B 0,C 180,E1 -411.761,E2 -411.761} C_VEL
LIN {X 0,Y 608.479,Z 278.837,A -85,B 0,C 180,E1 -414.42,E2 -414.42} C_VEL
LIN {X 0,Y 608.53,Z 287.365,A -85,B 0,C 180,E1 -416.73,E2 -416.73} C_VEL
LIN {X 0,Y 608.529,Z 297.85,A -85,B 0,C 180,E1 -419.458,E2 -419.458} C_VEL
LIN {X 0,Y 608.527,Z 309.624,A -85,B 0,C 180,E1 -422.486,E2 -422.486} C_VEL
LIN {X 0,Y 608.469,Z 319.876,A -85,B 0,C 180,E1 -425.065,E2 -425.065} C_VEL
LIN {X 0,Y 608.436,Z 330.127,A -85,B 0,C 180,E1 -427.593,E2 -427.593} C_VEL
LIN {X 0,Y 608.485,Z 340.378,A -85,B 0,C 180,E1 -430.079,E2 -430.079} C_VEL
LIN {X 0,Y 608.437,Z 352.094,A -85,B 0,C 180,E1 -432.869,E2 -432.869} C_VEL
LIN {X 0,Y 608.457,Z 363.81,A -85,B 0,C 180,E1 -435.621,E2 -435.621} C_VEL
LIN {X 0,Y 608.441,Z 374.976,A -85,B 0,C 180,E1 -438.211,E2 -438.211} C_VEL
LIN {X 0,Y 608.548,Z 389.091,A -85,B 0,C 180,E1 -438.488,E2 -438.488} C_VEL
LIN {X 0,Y 608.495,Z 401.472,A -85,B 0,C 180,E1 -438.863,E2 -438.863} C_VEL
LIN {X 0,Y 608.455,Z 413.171,A -85,B 0,C 180,E1 -439.35,E2 -439.35} C_VEL
LIN {X 0,Y 608.479,Z 425.577,A -85,B 0,C 180,E1 -440.023,E2 -440.023} C_VEL
LIN {X 0,Y 608.483,Z 436.473,A -85,B 0,C 180,E1 -440.778,E2 -440.778} C_VEL
LIN {X 0,Y 608.475,Z 447.111,A -85,B 0,C 180,E1 -441.699,E2 -441.699} C_VEL
LIN {X 0,Y 608.471,Z 454.96,A -85,B 0,C 180,E1 -442.534,E2 -442.534} C_VEL
LIN {X 0,Y 608.461,Z 462.286,A -85,B 0,C 180,E1 -443.484,E2 -443.484} C_VEL
LIN {X 0,Y 608.451,Z 467.866,A -85,B 0,C 180,E1 -444.366,E2 -444.366} C_VEL
LIN {X 0,Y 608.432,Z 472.95,A -85,B 0,C 180,E1 -445.362,E2 -445.362} C_VEL
LIN {X 0,Y 608.449,Z 476.896,A -85,B 0,C 180,E1 -446.358,E2 -446.358} C_VEL
LIN {X 0,Y 608.425,Z 479.809,A -85,B 0,C 180,E1 -447.352,E2 -447.352} C_VEL
LIN {X 0,Y 608.445,Z 481.201,A -85,B 0,C 180,E1 -448.014,E2 -448.014} C_VEL
LIN {X 0,Y 608.438,Z 482.783,A -85,B 0,C 180,E1 -449.338,E2 -449.338} C_VEL
LIN {X 0,Y 608.434,Z 483,A -85,B 0,C 180,E1 -450,E2 -450} C_VEL
LIN {X 0,Y 608.448,Z 482.184,A -85,B 0,C 180,E1 -451.324,E2 -451.324} C_VEL
LIN {X 0,Y 608.445,Z 481.201,A -85,B 0,C 180,E1 -451.986,E2 -451.986} C_VEL
LIN {X 0,Y 608.425,Z 479.809,A -85,B 0,C 180,E1 -452.648,E2 -452.648} C_VEL
LIN {X 0,Y 608.449,Z 476.896,A -85,B 0,C 180,E1 -453.642,E2 -453.642} C_VEL
LIN {X 0,Y 608.432,Z 472.95,A -85,B 0,C 180,E1 -454.638,E2 -454.638} C_VEL
LIN {X 0,Y 608.438,Z 466.876,A -85,B 0,C 180,E1 -455.801,E2 -455.801} C_VEL
LIN {X 0,Y 608.462,Z 460.234,A -85,B 0,C 180,E1 -456.799,E2 -456.799} C_VEL
LIN {X 0,Y 608.456,Z 451.988,A -85,B 0,C 180,E1 -457.8,E2 -457.8} C_VEL
LIN {X 0,Y 608.472,Z 443.535,A -85,B 0,C 180,E1 -458.636,E2 -458.636} C_VEL
LIN {X 0,Y 608.481,Z 433.089,A -85,B 0,C 180,E1 -459.473,E2 -459.473} C_VEL
LIN {X 0,Y 608.491,Z 422.754,A -85,B 0,C 180,E1 -460.145,E2 -460.145} C_VEL
LIN {X 0,Y 608.477,Z 411.347,A -85,B 0,C 180,E1 -460.737,E2 -460.737} C_VEL
LIN {X 0,Y 608.531,Z 399.006,A -85,B 0,C 180,E1 -461.221,E2 -461.221} C_VEL
LIN {X 0,Y 608.55,Z 385.433,A -85,B 0,C 180,E1 -461.597,E2 -461.597} C_VEL
LIN {X 0,Y 608.443,Z 374.976,A -85,B 0,C 180,E1 -461.789,E2 -461.789} C_VEL
LIN {X 0,Y 608.457,Z 363.81,A -85,B 0,C 180,E1 -464.379,E2 -464.379} C_VEL
LIN {X 0,Y 608.437,Z 352.094,A -85,B 0,C 180,E1 -467.131,E2 -467.131} C_VEL
LIN {X 0,Y 608.487,Z 340.378,A -85,B 0,C 180,E1 -469.921,E2 -469.921} C_VEL
LIN {X 0,Y 608.432,Z 329.872,A -85,B 0,C 180,E1 -472.469,E2 -472.469} C_VEL
LIN {X 0,Y 608.469,Z 319.876,A -85,B 0,C 180,E1 -474.935,E2 -474.935} C_VEL
LIN {X 0,Y 608.527,Z 309.624,A -85,B 0,C 180,E1 -477.514,E2 -477.514} C_VEL
LIN {X 0,Y 608.529,Z 297.825,A -85,B 0,C 180,E1 -480.542,E2 -480.542} C_VEL
LIN {X 0,Y 608.521,Z 287.161,A -85,B 0,C 180,E1 -483.271,E2 -483.271} C_VEL
LIN {X 0,Y 608.462,Z 278.695,A -85,B 0,C 180,E1 -485.556,E2 -485.556} C_VEL
LIN {X 0,Y 608.47,Z 278.694,A -85,B 0,C 180,E1 -488.24,E2 -488.24} C_VEL
LIN {X 0,Y 608.461,Z 278.695,A -85,B 0,C 180,E1 -491.342,E2 -491.342} C_VEL
LIN {X 0,Y 608.461,Z 278.695,A -85,B 0,C 180,E1 -494.264,E2 -494.264} C_VEL
LIN {X 0,Y 608.456,Z 278.698,A -85,B 0,C 180,E1 -497.04,E2 -497.04} C_VEL
LIN {X 0,Y 608.457,Z 278.695,A -85,B 0,C 180,E1 -499.697,E2 -499.697} C_VEL
LIN {X 0,Y 608.471,Z 278.694,A -85,B 0,C 180,E1 -502.254,E2 -502.254} C_VEL
LIN {X 0,Y 608.454,Z 278.698,A -85,B 0,C 180,E1 -505.095,E2 -505.095} C_VEL
LIN {X 0,Y 608.462,Z 278.696,A -85,B 0,C 180,E1 -507.905,E2 -507.905} C_VEL
LIN {X 0,Y 608.479,Z 278.694,A -85,B 0,C 180,E1 -510.221,E2 -510.221} C_VEL
LIN {X 0,Y 608.45,Z 278.697,A -85,B 0,C 180,E1 -513.226,E2 -513.226} C_VEL
LIN {X 0,Y 608.478,Z 278.693,A -85,B 0,C 180,E1 -515.849,E2 -515.849} C_VEL
LIN {X 0,Y 608.474,Z 278.694,A -85,B 0,C 180,E1 -518.308,E2 -518.308} C_VEL
LIN {X 0,Y 608.471,Z 278.694,A -85,B 0,C 180,E1 -521.286,E2 -521.286} C_VEL
LIN {X 0,Y 608.461,Z 278.696,A -85,B 0,C 180,E1 -523.906,E2 -523.906} C_VEL
LIN {X 0,Y 608.466,Z 278.694,A -85,B 0,C 180,E1 -526.644,E2 -526.644} C_VEL
LIN {X 0,Y 608.46,Z 278.695,A -85,B 0,C 180,E1 -529.35,E2 -529.35} C_VEL
LIN {X 0,Y 608.479,Z 278.694,A -85,B 0,C 180,E1 -532.033,E2 -532.033} C_VEL
LIN {X 0,Y 608.459,Z 278.695,A -85,B 0,C 180,E1 -534.698,E2 -534.698} C_VEL
LIN {X 0,Y 608.476,Z 278.694,A -85,B 0,C 180,E1 -537.352,E2 -537.352} C_VEL
LIN {X 0,Y 608.484,Z 278.693,A -85,B 0,C 180,E1 -540,E2 -540} C_VEL
LIN {X 0,Y 608.469,Z 278.694,A -85,B 0,C 180,E1 -542.648,E2 -542.648} C_VEL
LIN {X 0,Y 608.472,Z 278.695,A -85,B 0,C 180,E1 -545.302,E2 -545.302} C_VEL
LIN {X 0,Y 608.483,Z 278.693,A -85,B 0,C 180,E1 -547.967,E2 -547.967} C_VEL
LIN {X 0,Y 608.421,Z 278.929,A -85,B 0,C 180,E1 -549.445,E2 -549.445} C_VEL
LIN {X 0,Y 607.744,Z 279.611,A -85,B 0,C 180,E1 -549.994,E2 -549.994} C_VEL
LIN {X 0,Y 604.886,Z 280.82,A -85,B 0,C 180,E1 -550.883,E2 -550.883} C_VEL
LIN {X 0,Y 602.467,Z 281.798,A -85,B 0,C 180,E1 -551.599,E2 -551.599} C_VEL
LIN {X 0,Y 601.416,Z 282.507,A -85,B 0,C 180,E1 -552.151,E2 -552.151} C_VEL
LIN {X 0,Y 601.323,Z 282.733,A -85,B 0,C 180,E1 -552.338,E2 -552.338} C_VEL
LIN {X 0,Y 601.336,Z 285.794,A -85,B 0,C 180,E1 -554.899,E2 -554.899} C_VEL
LIN {X 0,Y 601.305,Z 289.199,A -85,B 0,C 180,E1 -557.691,E2 -557.691} C_VEL
LIN {X 0,Y 601.338,Z 292.716,A -85,B 0,C 180,E1 -560.525,E2 -560.525} C_VEL
LIN {X 0,Y 601.312,Z 296.362,A -85,B 0,C 180,E1 -563.415,E2 -563.415} C_VEL
LIN {X 0,Y 601.339,Z 299.906,A -85,B 0,C 180,E1 -566.188,E2 -566.188} C_VEL
LIN {X 0,Y 601.602,Z 307.724,A -85,B 0,C 180,E1 -566.366,E2 -566.366} C_VEL
LIN {X 0,Y 601.541,Z 320.195,A -85,B 0,C 180,E1 -566.731,E2 -566.731} C_VEL
LIN {X 0,Y 601.561,Z 331.634,A -85,B 0,C 180,E1 -567.197,E2 -567.197} C_VEL
LIN {X 0,Y 601.479,Z 342.867,A -85,B 0,C 180,E1 -567.787,E2 -567.787} C_VEL
LIN {X 0,Y 601.462,Z 354.049,A -85,B 0,C 180,E1 -568.53,E2 -568.53} C_VEL
LIN {X 0,Y 601.428,Z 362.604,A -85,B 0,C 180,E1 -569.226,E2 -569.226} C_VEL
LIN {X 0,Y 601.413,Z 372.095,A -85,B 0,C 180,E1 -570.165,E2 -570.165} C_VEL
LIN {X 0,Y 601.382,Z 380.461,A -85,B 0,C 180,E1 -571.196,E2 -571.196} C_VEL
LIN {X 0,Y 601.361,Z 387.742,A -85,B 0,C 180,E1 -572.322,E2 -572.322} C_VEL
LIN {X 0,Y 601.369,Z 392.796,A -85,B 0,C 180,E1 -573.317,E2 -573.317} C_VEL
LIN {X 0,Y 601.341,Z 397.434,A -85,B 0,C 180,E1 -574.529,E2 -574.529} C_VEL
LIN {X 0,Y 601.318,Z 400.666,A -85,B 0,C 180,E1 -575.759,E2 -575.759} C_VEL
LIN {X 0,Y 601.328,Z 402.048,A -85,B 0,C 180,E1 -576.588,E2 -576.588} C_VEL
LIN {X 0,Y 601.332,Z 402.819,A -85,B 0,C 180,E1 -577.427,E2 -577.427} C_VEL
LIN {X 0,Y 601.318,Z 402.911,A -85,B 0,C 180,E1 -578.456,E2 -578.456} C_VEL
LIN {X 0,Y 601.319,Z 402.025,A -85,B 0,C 180,E1 -579.521,E2 -579.521} C_VEL
LIN {X 0,Y 601.33,Z 399.397,A -85,B 0,C 180,E1 -580.881,E2 -580.881} C_VEL
LIN {X 0,Y 601.359,Z 395.273,A -85,B 0,C 180,E1 -582.176,E2 -582.176} C_VEL
LIN {X 0,Y 601.345,Z 390.041,A -85,B 0,C 180,E1 -583.343,E2 -583.343} C_VEL
LIN {X 0,Y 601.401,Z 383.065,A -85,B 0,C 180,E1 -584.52,E2 -584.52} C_VEL
LIN {X 0,Y 601.401,Z 375.941,A -85,B 0,C 180,E1 -585.479,E2 -585.479} C_VEL
LIN {X 0,Y 601.414,Z 367.275,A -85,B 0,C 180,E1 -586.429,E2 -586.429} C_VEL
LIN {X 0,Y 601.451,Z 357.011,A -85,B 0,C 180,E1 -587.333,E2 -587.333} C_VEL
LIN {X 0,Y 601.471,Z 347.534,A -85,B 0,C 180,E1 -588.014,E2 -588.014} C_VEL
LIN {X 0,Y 601.494,Z 335.888,A -85,B 0,C 180,E1 -588.688,E2 -588.688} C_VEL
LIN {X 0,Y 601.544,Z 323.853,A -85,B 0,C 180,E1 -589.222,E2 -589.222} C_VEL
LIN {X 0,Y 601.588,Z 310.695,A -85,B 0,C 180,E1 -589.65,E2 -589.65} C_VEL
LIN {X 0,Y 601.41,Z 300.908,A -85,B 0,C 180,E1 -589.873,E2 -589.873} C_VEL
LIN {X 0,Y 601.328,Z 299.901,A -85,B 0,C 180,E1 -589.906,E2 -589.906} C_VEL
LIN {X 0,Y 601.327,Z 296.417,A -85,B 0,C 180,E1 -592.632,E2 -592.632} C_VEL
LIN {X 0,Y 601.347,Z 293.345,A -85,B 0,C 180,E1 -595.063,E2 -595.063} C_VEL
LIN {X 0,Y 601.323,Z 290.336,A -85,B 0,C 180,E1 -597.477,E2 -597.477} C_VEL
LIN {X 0,Y 601.312,Z 287.396,A -85,B 0,C 180,E1 -599.871,E2 -599.871} C_VEL
LIN {X 0,Y 601.347,Z 284.041,A -85,B 0,C 180,E1 -602.65,E2 -602.65} C_VEL
LIN {X 0,Y 601.337,Z 281.126,A -85,B 0,C 180,E1 -605.118,E2 -605.118} C_VEL
LIN {X 0,Y 601.351,Z 279.582,A -85,B 0,C 180,E1 -606.587,E2 -606.587} C_VEL
LIN {X 0,Y 601.432,Z 279.572,A -85,B 0,C 180,E1 -609.478,E2 -609.478} C_VEL
LIN {X 0,Y 601.391,Z 279.576,A -85,B 0,C 180,E1 -612.311,E2 -612.311} C_VEL
LIN {X 0,Y 601.418,Z 279.57,A -85,B 0,C 180,E1 -614.409,E2 -614.409} C_VEL
LIN {X 0,Y 601.418,Z 279.572,A -85,B 0,C 180,E1 -617.172,E2 -617.172} C_VEL
LIN {X 0,Y 601.434,Z 279.571,A -85,B 0,C 180,E1 -619.905,E2 -619.905} C_VEL
LIN {X 0,Y 601.441,Z 279.571,A -85,B 0,C 180,E1 -622.615,E2 -622.615} C_VEL
LIN {X 0,Y 601.425,Z 279.573,A -85,B 0,C 180,E1 -625.308,E2 -625.308} C_VEL
LIN {X 0,Y 601.436,Z 279.572,A -85,B 0,C 180,E1 -627.991,E2 -627.991} C_VEL
LIN {X 0,Y 601.449,Z 279.569,A -85,B 0,C 180,E1 -630.67,E2 -630.67} C_VEL
LIN {X 0,Y 601.437,Z 279.57,A -85,B 0,C 180,E1 -633.35,E2 -633.35} C_VEL
LIN {X 0,Y 601.415,Z 279.572,A -85,B 0,C 180,E1 -636.037,E2 -636.037} C_VEL
LIN {X 0,Y 601.443,Z 279.568,A -85,B 0,C 180,E1 -638.061,E2 -638.061} C_VEL
LIN {X 0,Y 601.42,Z 279.574,A -85,B 0,C 180,E1 -641.009,E2 -641.009} C_VEL
LIN {X 0,Y 601.402,Z 279.575,A -85,B 0,C 180,E1 -643.516,E2 -643.516} C_VEL
LIN {X 0,Y 601.441,Z 279.572,A -85,B 0,C 180,E1 -646.287,E2 -646.287} C_VEL
LIN {X 0,Y 601.418,Z 279.572,A -85,B 0,C 180,E1 -649.099,E2 -649.099} C_VEL
LIN {X 0,Y 601.401,Z 279.573,A -85,B 0,C 180,E1 -651.24,E2 -651.24} C_VEL
LIN {X 0,Y 601.461,Z 279.569,A -85,B 0,C 180,E1 -654.14,E2 -654.14} C_VEL
LIN {X 0,Y 601.455,Z 279.566,A -85,B 0,C 180,E1 -657.111,E2 -657.111} C_VEL
LIN {X 0,Y 601.397,Z 279.577,A -85,B 0,C 180,E1 -659.395,E2 -659.395} C_VEL
LIN {X 0,Y 601.413,Z 279.572,A -85,B 0,C 180,E1 -661.727,E2 -661.727} C_VEL
LIN {X 0,Y 601.42,Z 279.57,A -85,B 0,C 180,E1 -664.119,E2 -664.119} C_VEL
LIN {X 0,Y 601.4,Z 279.572,A -85,B 0,C 180,E1 -666.584,E2 -666.584} C_VEL
LIN {X 0,Y 601.444,Z 279.567,A -85,B 0,C 180,E1 -669.536,E2 -669.536} C_VEL
LIN {X 0,Y 601.412,Z 279.575,A -85,B 0,C 180,E1 -672.591,E2 -672.591} C_VEL
LIN {X 0,Y 601.401,Z 279.573,A -85,B 0,C 180,E1 -675.48,E2 -675.48} C_VEL
LIN {X 0,Y 601.424,Z 279.569,A -85,B 0,C 180,E1 -678.407,E2 -678.407} C_VEL
LIN {X 0,Y 601.439,Z 279.568,A -85,B 0,C 180,E1 -680.876,E2 -680.876} C_VEL
LIN {X 0,Y 601.404,Z 279.573,A -85,B 0,C 180,E1 -683.417,E2 -683.417} C_VEL
LIN {X 0,Y 601.419,Z 279.57,A -85,B 0,C 180,E1 -686.067,E2 -686.067} C_VEL
LIN {X 0,Y 601.416,Z 279.57,A -85,B 0,C 180,E1 -689.058,E2 -689.058} C_VEL
LIN {X 0,Y 601.413,Z 279.571,A -85,B 0,C 180,E1 -691.372,E2 -691.372} C_VEL
LIN {X 0,Y 601.402,Z 279.575,A -85,B 0,C 180,E1 -693.636,E2 -693.636} C_VEL
LIN {X 0,Y 601.399,Z 279.573,A -85,B 0,C 180,E1 -696.589,E2 -696.589} C_VEL
LIN {X 0,Y 601.423,Z 279.57,A -85,B 0,C 180,E1 -699.205,E2 -699.205} C_VEL
LIN {X 0,Y 601.423,Z 279.572,A -85,B 0,C 180,E1 -701.608,E2 -701.608} C_VEL
LIN {X 0,Y 601.41,Z 279.572,A -85,B 0,C 180,E1 -704.409,E2 -704.409} C_VEL
LIN {X 0,Y 601.407,Z 279.572,A -85,B 0,C 180,E1 -707.172,E2 -707.172} C_VEL
LIN {X 0,Y 601.439,Z 279.567,A -85,B 0,C 180,E1 -709.905,E2 -709.905} C_VEL
LIN {X 0,Y 601.411,Z 279.571,A -85,B 0,C 180,E1 -712.615,E2 -712.615} C_VEL
LIN {X 0,Y 601.404,Z 279.572,A -85,B 0,C 180,E1 -715.308,E2 -715.308} C_VEL
LIN {X 0,Y 601.438,Z 279.567,A -85,B 0,C 180,E1 -717.991,E2 -717.991} C_VEL
LIN {X 0,Y 601.442,Z 279.567,A -85,B 0,C 180,E1 -720.67,E2 -720.67} C_VEL
LIN {X 0,Y 601.385,Z 279.575,A -85,B 0,C 180,E1 -723.35,E2 -723.35} C_VEL
LIN {X 0,Y 601.419,Z 279.571,A -85,B 0,C 180,E1 -726.037,E2 -726.037} C_VEL
LIN {X 0,Y 601.409,Z 279.573,A -85,B 0,C 180,E1 -728.738,E2 -728.738} C_VEL
LIN {X 0,Y 601.412,Z 279.573,A -85,B 0,C 180,E1 -731.459,E2 -731.459} C_VEL
LIN {X 0,Y 601.42,Z 279.574,A -85,B 0,C 180,E1 -734.206,E2 -734.206} C_VEL
LIN {X 0,Y 601.417,Z 279.573,A -85,B 0,C 180,E1 -736.986,E2 -736.986} C_VEL
LIN {X 0,Y 601.396,Z 279.574,A -85,B 0,C 180,E1 -739.81,E2 -739.81} C_VEL
LIN {X 0,Y 601.414,Z 279.571,A -85,B 0,C 180,E1 -742.604,E2 -742.604} C_VEL
LIN {X 0,Y 601.4,Z 279.575,A -85,B 0,C 180,E1 -744.879,E2 -744.879} C_VEL
LIN {X 0,Y 601.394,Z 279.573,A -85,B 0,C 180,E1 -747.869,E2 -747.869} C_VEL
LIN {X 0,Y 601.41,Z 279.573,A -85,B 0,C 180,E1 -750.165,E2 -750.165} C_VEL
LIN {X 0,Y 601.422,Z 279.573,A -85,B 0,C 180,E1 -752.715,E2 -752.715} C_VEL
LIN {X 0,Y 601.382,Z 279.577,A -85,B 0,C 180,E1 -755.109,E2 -755.109} C_VEL
LIN {X 0,Y 601.44,Z 279.567,A -85,B 0,C 180,E1 -757.419,E2 -757.419} C_VEL
LIN {X 0,Y 601.403,Z 279.572,A -85,B 0,C 180,E1 -759.996,E2 -759.996} C_VEL
LIN {X 0,Y 601.39,Z 279.574,A -85,B 0,C 180,E1 -762.672,E2 -762.672} C_VEL
LIN {X 0,Y 601.431,Z 279.57,A -85,B 0,C 180,E1 -765.482,E2 -765.482} C_VEL
LIN {X 0,Y 601.424,Z 279.573,A -85,B 0,C 180,E1 -768.407,E2 -768.407} C_VEL
LIN {X 0,Y 601.41,Z 279.574,A -85,B 0,C 180,E1 -770.873,E2 -770.873} C_VEL
LIN {X 0,Y 601.405,Z 279.575,A -85,B 0,C 180,E1 -773.417,E2 -773.417} C_VEL
LIN {X 0,Y 601.432,Z 279.676,A -85,B 0,C 180,E1 -774.203,E2 -774.203} C_VEL
LIN {X 0,Y 601.617,Z 285.745,A -85,B 0,C 180,E1 -775.893,E2 -775.893} C_VEL
LIN {X 0,Y 601.548,Z 296.62,A -85,B 0,C 180,E1 -778.793,E2 -778.793} C_VEL
LIN {X 0,Y 601.556,Z 308.16,A -85,B 0,C 180,E1 -781.76,E2 -781.76} C_VEL
LIN {X 0,Y 601.496,Z 318.411,A -85,B 0,C 180,E1 -784.385,E2 -784.385} C_VEL
LIN {X 0,Y 601.43,Z 328.662,A -85,B 0,C 180,E1 -786.954,E2 -786.954} C_VEL
LIN {X 0,Y 601.407,Z 338.914,A -85,B 0,C 180,E1 -789.477,E2 -789.477} C_VEL
LIN {X 0,Y 601.426,Z 350.63,A -85,B 0,C 180,E1 -792.312,E2 -792.312} C_VEL
LIN {X 0,Y 601.379,Z 362.345,A -85,B 0,C 180,E1 -795.102,E2 -795.102} C_VEL
LIN {X 0,Y 601.366,Z 372.597,A -85,B 0,C 180,E1 -797.514,E2 -797.514} C_VEL
LIN {X 0,Y 601.38,Z 374.976,A -85,B 0,C 180,E1 -798.071,E2 -798.071} C_VEL
LIN {X 0,Y 601.609,Z 387.263,A -85,B 0,C 180,E1 -798.31,E2 -798.31} C_VEL
LIN {X 0,Y 601.564,Z 400.292,A -85,B 0,C 180,E1 -798.69,E2 -798.69} C_VEL
LIN {X 0,Y 601.495,Z 411.805,A -85,B 0,C 180,E1 -799.159,E2 -799.159} C_VEL
LIN {X 0,Y 601.47,Z 424.167,A -85,B 0,C 180,E1 -799.82,E2 -799.82} C_VEL
LIN {X 0,Y 601.455,Z 435.402,A -85,B 0,C 180,E1 -800.585,E2 -800.585} C_VEL
LIN {X 0,Y 601.423,Z 445.336,A -85,B 0,C 180,E1 -801.431,E2 -801.431} C_VEL
LIN {X 0,Y 601.418,Z 454.96,A -85,B 0,C 180,E1 -802.446,E2 -802.446} C_VEL
LIN {X 0,Y 601.37,Z 462.225,A -85,B 0,C 180,E1 -803.398,E2 -803.398} C_VEL
LIN {X 0,Y 601.372,Z 467.866,A -85,B 0,C 180,E1 -804.299,E2 -804.299} C_VEL
LIN {X 0,Y 601.336,Z 472.95,A -85,B 0,C 180,E1 -805.307,E2 -805.307} C_VEL
LIN {X 0,Y 601.368,Z 476.896,A -85,B 0,C 180,E1 -806.315,E2 -806.315} C_VEL
LIN {X 0,Y 601.325,Z 479.809,A -85,B 0,C 180,E1 -807.32,E2 -807.32} C_VEL
LIN {X 0,Y 601.343,Z 481.202,A -85,B 0,C 180,E1 -807.991,E2 -807.991} C_VEL
LIN {X 0,Y 601.339,Z 482.784,A -85,B 0,C 180,E1 -809.33,E2 -809.33} C_VEL
LIN {X 0,Y 601.335,Z 483,A -85,B 0,C 180,E1 -810,E2 -810} C_VEL
LIN {X 0,Y 601.347,Z 482.184,A -85,B 0,C 180,E1 -811.339,E2 -811.339} C_VEL
LIN {X 0,Y 601.343,Z 481.202,A -85,B 0,C 180,E1 -812.009,E2 -812.009} C_VEL
LIN {X 0,Y 601.325,Z 479.809,A -85,B 0,C 180,E1 -812.68,E2 -812.68} C_VEL
LIN {X 0,Y 601.368,Z 476.896,A -85,B 0,C 180,E1 -813.685,E2 -813.685} C_VEL
LIN {X 0,Y 601.336,Z 472.95,A -85,B 0,C 180,E1 -814.693,E2 -814.693} C_VEL
LIN {X 0,Y 601.373,Z 466.877,A -85,B 0,C 180,E1 -815.869,E2 -815.869} C_VEL
LIN {X 0,Y 601.382,Z 460.235,A -85,B 0,C 180,E1 -816.88,E2 -816.88} C_VEL
LIN {X 0,Y 601.4,Z 451.989,A -85,B 0,C 180,E1 -817.892,E2 -817.892} C_VEL
LIN {X 0,Y 601.436,Z 443.536,A -85,B 0,C 180,E1 -818.738,E2 -818.738} C_VEL
LIN {X 0,Y 601.449,Z 433.091,A -85,B 0,C 180,E1 -819.585,E2 -819.585} C_VEL
LIN {X 0,Y 601.482,Z 422.755,A -85,B 0,C 180,E1 -820.264,E2 -820.264} C_VEL
LIN {X 0,Y 601.493,Z 411.118,A -85,B 0,C 180,E1 -820.874,E2 -820.874} C_VEL
LIN {X 0,Y 601.56,Z 398.311,A -85,B 0,C 180,E1 -821.376,E2 -821.376} C_VEL
LIN {X 0,Y 601.599,Z 385.433,A -85,B 0,C 180,E1 -821.733,E2 -821.733} C_VEL
LIN {X 0,Y 601.382,Z 374.976,A -85,B 0,C 180,E1 -821.929,E2 -821.929} C_VEL
LIN {X 0,Y 601.396,Z 363.81,A -85,B 0,C 180,E1 -824.552,E2 -824.552} C_VEL
LIN {X 0,Y 601.405,Z 352.094,A -85,B 0,C 180,E1 -827.337,E2 -827.337} C_VEL
LIN {X 0,Y 601.423,Z 340.378,A -85,B 0,C 180,E1 -830.165,E2 -830.165} C_VEL
LIN {X 0,Y 601.404,Z 330.127,A -85,B 0,C 180,E1 -832.684,E2 -832.684} C_VEL
LIN {X 0,Y 601.503,Z 319.876,A -85,B 0,C 180,E1 -835.244,E2 -835.244} C_VEL
LIN {X 0,Y 601.55,Z 309.624,A -85,B 0,C 180,E1 -837.861,E2 -837.861} C_VEL
LIN {X 0,Y 601.523,Z 300.539,A -85,B 0,C 180,E1 -840.163,E2 -840.163} C_VEL
LIN {X 0,Y 601.561,Z 289.647,A -85,B 0,C 180,E1 -842.982,E2 -842.982} C_VEL
LIN {X 0,Y 601.59,Z 280.745,A -85,B 0,C 180,E1 -845.401,E2 -845.401} C_VEL
LIN {X 0,Y 601.425,Z 279.573,A -85,B 0,C 180,E1 -845.752,E2 -845.752} C_VEL
LIN {X 0,Y 601.437,Z 279.57,A -85,B 0,C 180,E1 -848.471,E2 -848.471} C_VEL
LIN {X 0,Y 601.427,Z 279.571,A -85,B 0,C 180,E1 -851.593,E2 -851.593} C_VEL
LIN {X 0,Y 601.43,Z 279.571,A -85,B 0,C 180,E1 -854.535,E2 -854.535} C_VEL
LIN {X 0,Y 601.412,Z 279.573,A -85,B 0,C 180,E1 -857.41,E2 -857.41} C_VEL
LIN {X 0,Y 601.445,Z 279.569,A -85,B 0,C 180,E1 -860.464,E2 -860.464} C_VEL
LIN {X 0,Y 601.408,Z 279.573,A -85,B 0,C 180,E1 -863.417,E2 -863.417} C_VEL
LIN {X 0,Y 601.437,Z 279.572,A -85,B 0,C 180,E1 -866.065,E2 -866.065} C_VEL
LIN {X 0,Y 601.436,Z 279.572,A -85,B 0,C 180,E1 -869.059,E2 -869.059} C_VEL
LIN {X 0,Y 601.429,Z 279.571,A -85,B 0,C 180,E1 -871.373,E2 -871.373} C_VEL
LIN {X 0,Y 601.404,Z 279.574,A -85,B 0,C 180,E1 -873.636,E2 -873.636} C_VEL
LIN {X 0,Y 601.424,Z 279.571,A -85,B 0,C 180,E1 -876.59,E2 -876.59} C_VEL
LIN {X 0,Y 601.429,Z 279.571,A -85,B 0,C 180,E1 -879.478,E2 -879.478} C_VEL
LIN {X 0,Y 601.402,Z 279.575,A -85,B 0,C 180,E1 -882.312,E2 -882.312} C_VEL
LIN {X 0,Y 601.416,Z 279.572,A -85,B 0,C 180,E1 -884.409,E2 -884.409} C_VEL
LIN {X 0,Y 601.416,Z 279.574,A -85,B 0,C 180,E1 -887.172,E2 -887.172} C_VEL
LIN {X 0,Y 601.44,Z 279.57,A -85,B 0,C 180,E1 -889.905,E2 -889.905} C_VEL
LIN {X 0,Y 601.414,Z 279.572,A -85,B 0,C 180,E1 -892.614,E2 -892.614} C_VEL
LIN {X 0,Y 601.419,Z 279.573,A -85,B 0,C 180,E1 -895.308,E2 -895.308} C_VEL
LIN {X 0,Y 601.438,Z 279.571,A -85,B 0,C 180,E1 -897.991,E2 -897.991} C_VEL
LIN {X 0,Y 601.446,Z 279.568,A -85,B 0,C 180,E1 -900.669,E2 -900.669} C_VEL
LIN {X 0,Y 601.437,Z 279.57,A -85,B 0,C 180,E1 -903.349,E2 -903.349} C_VEL
LIN {X 0,Y 601.419,Z 279.573,A -85,B 0,C 180,E1 -906.037,E2 -906.037} C_VEL
LIN {X 0,Y 601.445,Z 279.57,A -85,B 0,C 180,E1 -908.061,E2 -908.061} C_VEL
LIN {X 0,Y 601.354,Z 279.596,A -85,B 0,C 180,E1 -909.434,E2 -909.434} C_VEL
LIN {X 0,Y 601.336,Z 281.698,A -85,B 0,C 180,E1 -911.46,E2 -911.46} C_VEL
LIN {X 0,Y 601.323,Z 282.733,A -85,B 0,C 180,E1 -912.338,E2 -912.338} C_VEL
LIN {X 0,Y 600.638,Z 283.428,A -85,B 0,C 180,E1 -912.894,E2 -912.894} C_VEL
LIN {X 0,Y 597.78,Z 284.648,A -85,B 0,C 180,E1 -913.794,E2 -913.794} C_VEL
LIN {X 0,Y 595.373,Z 285.633,A -85,B 0,C 180,E1 -914.519,E2 -914.519} C_VEL
LIN {X 0,Y 594.335,Z 286.351,A -85,B 0,C 180,E1 -915.078,E2 -915.078} C_VEL
LIN {X 0,Y 594.247,Z 286.582,A -85,B 0,C 180,E1 -915.267,E2 -915.267} C_VEL
LIN {X 0,Y 594.204,Z 289.774,A -85,B 0,C 180,E1 -917.91,E2 -917.91} C_VEL
LIN {X 0,Y 594.241,Z 293.423,A -85,B 0,C 180,E1 -920.88,E2 -920.88} C_VEL
LIN {X 0,Y 594.212,Z 296.033,A -85,B 0,C 180,E1 -922.973,E2 -922.973} C_VEL
LIN {X 0,Y 594.225,Z 299.836,A -85,B 0,C 180,E1 -925.99,E2 -925.99} C_VEL
LIN {X 0,Y 594.228,Z 299.909,A -85,B 0,C 180,E1 -926.047,E2 -926.047} C_VEL
LIN {X 0,Y 594.624,Z 305.328,A -85,B 0,C 180,E1 -926.17,E2 -926.17} C_VEL
LIN {X 0,Y 594.596,Z 318.268,A -85,B 0,C 180,E1 -926.533,E2 -926.533} C_VEL
LIN {X 0,Y 594.562,Z 330.677,A -85,B 0,C 180,E1 -927.023,E2 -927.023} C_VEL
LIN {X 0,Y 594.482,Z 342.396,A -85,B 0,C 180,E1 -927.637,E2 -927.637} C_VEL
LIN {X 0,Y 594.447,Z 354.038,A -85,B 0,C 180,E1 -928.416,E2 -928.416} C_VEL
LIN {X 0,Y 594.383,Z 364.454,A -85,B 0,C 180,E1 -929.289,E2 -929.289} C_VEL
LIN {X 0,Y 594.349,Z 374.274,A -85,B 0,C 180,E1 -930.321,E2 -930.321} C_VEL
LIN {X 0,Y 594.305,Z 382.159,A -85,B 0,C 180,E1 -931.354,E2 -931.354} C_VEL
LIN {X 0,Y 594.269,Z 389.184,A -85,B 0,C 180,E1 -932.523,E2 -932.523} C_VEL
LIN {X 0,Y 594.269,Z 394.914,A -85,B 0,C 180,E1 -933.768,E2 -933.768} C_VEL
LIN {X 0,Y 594.255,Z 397.749,A -85,B 0,C 180,E1 -934.588,E2 -934.588} C_VEL
LIN {X 0,Y 594.229,Z 400,A -85,B 0,C 180,E1 -935.417,E2 -935.417} C_VEL
LIN {X 0,Y 594.222,Z 401.918,A -85,B 0,C 180,E1 -936.461,E2 -936.461} C_VEL
LIN {X 0,Y 594.229,Z 402.901,A -85,B 0,C 180,E1 -937.588,E2 -937.588} C_VEL
LIN {X 0,Y 594.21,Z 402.718,A -85,B 0,C 180,E1 -938.819,E2 -938.819} C_VEL
LIN {X 0,Y 594.231,Z 401.723,A -85,B 0,C 180,E1 -939.757,E2 -939.757} C_VEL
LIN {X 0,Y 594.231,Z 399.685,A -85,B 0,C 180,E1 -940.805,E2 -940.805} C_VEL
LIN {X 0,Y 594.263,Z 395.78,A -85,B 0,C 180,E1 -942.086,E2 -942.086} C_VEL
LIN {X 0,Y 594.276,Z 390.539,A -85,B 0,C 180,E1 -943.308,E2 -943.308} C_VEL
LIN {X 0,Y 594.309,Z 385.341,A -85,B 0,C 180,E1 -944.243,E2 -944.243} C_VEL
LIN {X 0,Y 594.31,Z 377.767,A -85,B 0,C 180,E1 -945.339,E2 -945.339} C_VEL
LIN {X 0,Y 594.346,Z 369.514,A -85,B 0,C 180,E1 -946.297,E2 -946.297} C_VEL
LIN {X 0,Y 594.385,Z 359.641,A -85,B 0,C 180,E1 -947.231,E2 -947.231} C_VEL
LIN {X 0,Y 594.458,Z 348.547,A -85,B 0,C 180,E1 -948.064,E2 -948.064} C_VEL
LIN {X 0,Y 594.497,Z 337.75,A -85,B 0,C 180,E1 -948.715,E2 -948.715} C_VEL
LIN {X 0,Y 594.583,Z 326.017,A -85,B 0,C 180,E1 -949.27,E2 -949.27} C_VEL
LIN {X 0,Y 594.614,Z 313.343,A -85,B 0,C 180,E1 -949.712,E2 -949.712} C_VEL
LIN {X 0,Y 594.526,Z 302.006,A -85,B 0,C 180,E1 -949.991,E2 -949.991} C_VEL
LIN {X 0,Y 594.218,Z 299.904,A -85,B 0,C 180,E1 -950.047,E2 -950.047} C_VEL
LIN {X 0,Y 594.217,Z 296.304,A -85,B 0,C 180,E1 -952.901,E2 -952.901} C_VEL
LIN {X 0,Y 594.233,Z 292.591,A -85,B 0,C 180,E1 -955.883,E2 -955.883} C_VEL
LIN {X 0,Y 594.244,Z 289.211,A -85,B 0,C 180,E1 -958.642,E2 -958.642} C_VEL
LIN {X 0,Y 594.232,Z 285.459,A -85,B 0,C 180,E1 -961.765,E2 -961.765} C_VEL
LIN {X 0,Y 594.226,Z 282.772,A -85,B 0,C 180,E1 -964.049,E2 -964.049} C_VEL
LIN {X 0,Y 594.25,Z 280.467,A -85,B 0,C 180,E1 -966.29,E2 -966.29} C_VEL
LIN {X 0,Y 594.361,Z 280.451,A -85,B 0,C 180,E1 -968.496,E2 -968.496} C_VEL
LIN {X 0,Y 594.377,Z 280.449,A -85,B 0,C 180,E1 -971.073,E2 -971.073} C_VEL
LIN {X 0,Y 594.411,Z 280.447,A -85,B 0,C 180,E1 -973.515,E2 -973.515} C_VEL
LIN {X 0,Y 594.379,Z 280.449,A -85,B 0,C 180,E1 -976.321,E2 -976.321} C_VEL
LIN {X 0,Y 594.363,Z 280.45,A -85,B 0,C 180,E1 -979.094,E2 -979.094} C_VEL
LIN {X 0,Y 594.417,Z 280.442,A -85,B 0,C 180,E1 -981.843,E2 -981.843} C_VEL
LIN {X 0,Y 594.382,Z 280.446,A -85,B 0,C 180,E1 -984.572,E2 -984.572} C_VEL
LIN {X 0,Y 594.392,Z 280.445,A -85,B 0,C 180,E1 -987.289,E2 -987.289} C_VEL
LIN {X 0,Y 594.418,Z 280.442,A -85,B 0,C 180,E1 -990,E2 -990} C_VEL
LIN {X 0,Y 594.396,Z 280.445,A -85,B 0,C 180,E1 -992.711,E2 -992.711} C_VEL
LIN {X 0,Y 594.379,Z 280.448,A -85,B 0,C 180,E1 -995.428,E2 -995.428} C_VEL
LIN {X 0,Y 594.415,Z 280.444,A -85,B 0,C 180,E1 -998.157,E2 -998.157} C_VEL
LIN {X 0,Y 594.385,Z 280.45,A -85,B 0,C 180,E1 -1001.07,E2 -1001.07} C_VEL
LIN {X 0,Y 594.366,Z 280.453,A -85,B 0,C 180,E1 -1003.679,E2 -1003.679} C_VEL
LIN {X 0,Y 594.375,Z 280.448,A -85,B 0,C 180,E1 -1006.713,E2 -1006.713} C_VEL
LIN {X 0,Y 594.369,Z 280.448,A -85,B 0,C 180,E1 -1009.335,E2 -1009.335} C_VEL
LIN {X 0,Y 594.358,Z 280.453,A -85,B 0,C 180,E1 -1011.504,E2 -1011.504} C_VEL
LIN {X 0,Y 594.391,Z 280.447,A -85,B 0,C 180,E1 -1014.446,E2 -1014.446} C_VEL
LIN {X 0,Y 594.383,Z 280.45,A -85,B 0,C 180,E1 -1016.7,E2 -1016.7} C_VEL
LIN {X 0,Y 594.375,Z 280.448,A -85,B 0,C 180,E1 -1018.999,E2 -1018.999} C_VEL
LIN {X 0,Y 594.393,Z 280.445,A -85,B 0,C 180,E1 -1021.645,E2 -1021.645} C_VEL
LIN {X 0,Y 594.382,Z 280.45,A -85,B 0,C 180,E1 -1024.58,E2 -1024.58} C_VEL
LIN {X 0,Y 594.388,Z 280.447,A -85,B 0,C 180,E1 -1027.608,E2 -1027.608} C_VEL
LIN {X 0,Y 594.367,Z 280.448,A -85,B 0,C 180,E1 -1030.568,E2 -1030.568} C_VEL
LIN {X 0,Y 594.369,Z 280.448,A -85,B 0,C 180,E1 -1033.3,E2 -1033.3} C_VEL
LIN {X 0,Y 594.362,Z 280.45,A -85,B 0,C 180,E1 -1036.162,E2 -1036.162} C_VEL
LIN {X 0,Y 594.381,Z 280.446,A -85,B 0,C 180,E1 -1038.536,E2 -1038.536} C_VEL
LIN {X 0,Y 594.39,Z 280.446,A -85,B 0,C 180,E1 -1041.296,E2 -1041.296} C_VEL
LIN {X 0,Y 594.352,Z 280.45,A -85,B 0,C 180,E1 -1043.756,E2 -1043.756} C_VEL
LIN {X 0,Y 594.367,Z 280.448,A -85,B 0,C 180,E1 -1046.238,E2 -1046.238} C_VEL
LIN {X 0,Y 594.373,Z 280.448,A -85,B 0,C 180,E1 -1048.65,E2 -1048.65} C_VEL
LIN {X 0,Y 594.379,Z 280.45,A -85,B 0,C 180,E1 -1051.044,E2 -1051.044} C_VEL
LIN {X 0,Y 594.384,Z 280.446,A -85,B 0,C 180,E1 -1053.979,E2 -1053.979} C_VEL
LIN {X 0,Y 594.367,Z 280.451,A -85,B 0,C 180,E1 -1056.295,E2 -1056.295} C_VEL
LIN {X 0,Y 594.392,Z 280.446,A -85,B 0,C 180,E1 -1059.224,E2 -1059.224} C_VEL
LIN {X 0,Y 594.357,Z 280.449,A -85,B 0,C 180,E1 -1062.095,E2 -1062.095} C_VEL
LIN {X 0,Y 594.373,Z 280.448,A -85,B 0,C 180,E1 -1064.922,E2 -1064.922} C_VEL
LIN {X 0,Y 594.389,Z 280.447,A -85,B 0,C 180,E1 -1067.712,E2 -1067.712} C_VEL
LIN {X 0,Y 594.37,Z 280.451,A -85,B 0,C 180,E1 -1070.471,E2 -1070.471} C_VEL
LIN {X 0,Y 594.406,Z 280.447,A -85,B 0,C 180,E1 -1073.309,E2 -1073.309} C_VEL
LIN {X 0,Y 594.361,Z 280.453,A -85,B 0,C 180,E1 -1075.932,E2 -1075.932} C_VEL
LIN {X 0,Y 594.407,Z 280.443,A -85,B 0,C 180,E1 -1077.967,E2 -1077.967} C_VEL
LIN {X 0,Y 594.414,Z 280.443,A -85,B 0,C 180,E1 -1080.678,E2 -1080.678} C_VEL
LIN {X 0,Y 594.34,Z 280.453,A -85,B 0,C 180,E1 -1083.39,E2 -1083.39} C_VEL
LIN {X 0,Y 594.369,Z 280.449,A -85,B 0,C 180,E1 -1086.109,E2 -1086.109} C_VEL
LIN {X 0,Y 594.378,Z 280.45,A -85,B 0,C 180,E1 -1088.842,E2 -1088.842} C_VEL
LIN {X 0,Y 594.381,Z 280.451,A -85,B 0,C 180,E1 -1091.596,E2 -1091.596} C_VEL
LIN {X 0,Y 594.388,Z 280.449,A -85,B 0,C 180,E1 -1094.377,E2 -1094.377} C_VEL
LIN {X 0,Y 594.383,Z 280.447,A -85,B 0,C 180,E1 -1097.194,E2 -1097.194} C_VEL
LIN {X 0,Y 594.368,Z 280.448,A -85,B 0,C 180,E1 -1100.054,E2 -1100.054} C_VEL
LIN {X 0,Y 594.361,Z 280.449,A -85,B 0,C 180,E1 -1102.733,E2 -1102.733} C_VEL
LIN {X 0,Y 594.377,Z 280.447,A -85,B 0,C 180,E1 -1105.193,E2 -1105.193} C_VEL
LIN {X 0,Y 594.353,Z 280.453,A -85,B 0,C 180,E1 -1107.519,E2 -1107.519} C_VEL
LIN {X 0,Y 594.373,Z 280.449,A -85,B 0,C 180,E1 -1109.777,E2 -1109.777} C_VEL
LIN {X 0,Y 594.364,Z 280.449,A -85,B 0,C 180,E1 -1112.148,E2 -1112.148} C_VEL
LIN {X 0,Y 594.373,Z 280.447,A -85,B 0,C 180,E1 -1114.581,E2 -1114.581} C_VEL
LIN {X 0,Y 594.393,Z 280.446,A -85,B 0,C 180,E1 -1117.608,E2 -1117.608} C_VEL
LIN {X 0,Y 594.368,Z 280.452,A -85,B 0,C 180,E1 -1120.567,E2 -1120.567} C_VEL
LIN {X 0,Y 594.364,Z 280.451,A -85,B 0,C 180,E1 -1123.3,E2 -1123.3} C_VEL
LIN {X 0,Y 594.371,Z 280.448,A -85,B 0,C 180,E1 -1126.16,E2 -1126.16} C_VEL
LIN {X 0,Y 594.381,Z 280.447,A -85,B 0,C 180,E1 -1129.178,E2 -1129.178} C_VEL
LIN {X 0,Y 594.381,Z 280.449,A -85,B 0,C 180,E1 -1132.059,E2 -1132.059} C_VEL
LIN {X 0,Y 594.371,Z 280.457,A -85,B 0,C 180,E1 -1133.966,E2 -1133.966} C_VEL
LIN {X 0,Y 594.655,Z 284.174,A -85,B 0,C 180,E1 -1135.034,E2 -1135.034} C_VEL
LIN {X 0,Y 594.629,Z 294.517,A -85,B 0,C 180,E1 -1137.868,E2 -1137.868} C_VEL
LIN {X 0,Y 594.552,Z 304.991,A -85,B 0,C 180,E1 -1140.623,E2 -1140.623} C_VEL
LIN {X 0,Y 594.532,Z 315.482,A -85,B 0,C 180,E1 -1143.307,E2 -1143.307} C_VEL
LIN {X 0,Y 594.445,Z 325.734,A -85,B 0,C 180,E1 -1145.928,E2 -1145.928} C_VEL
LIN {X 0,Y 594.431,Z 337.34,A -85,B 0,C 180,E1 -1148.835,E2 -1148.835} C_VEL
LIN {X 0,Y 594.394,Z 349.165,A -85,B 0,C 180,E1 -1151.74,E2 -1151.74} C_VEL
LIN {X 0,Y 594.333,Z 360.881,A -85,B 0,C 180,E1 -1154.57,E2 -1154.57} C_VEL
LIN {X 0,Y 594.316,Z 372.597,A -85,B 0,C 180,E1 -1157.363,E2 -1157.363} C_VEL
LIN {X 0,Y 594.293,Z 374.976,A -85,B 0,C 180,E1 -1157.926,E2 -1157.926} C_VEL
LIN {X 0,Y 594.688,Z 380.083,A -85,B 0,C 180,E1 -1158.021,E2 -1158.021} C_VEL
LIN {X 0,Y 594.63,Z 393.733,A -85,B 0,C 180,E1 -1158.344,E2 -1158.344} C_VEL
LIN {X 0,Y 594.541,Z 406.553,A -85,B 0,C 180,E1 -1158.797,E2 -1158.797} C_VEL
LIN {X 0,Y 594.481,Z 418.208,A -85,B 0,C 180,E1 -1159.355,E2 -1159.355} C_VEL
LIN {X 0,Y 594.466,Z 429.476,A -85,B 0,C 180,E1 -1160.043,E2 -1160.043} C_VEL
LIN {X 0,Y 594.406,Z 439.646,A -85,B 0,C 180,E1 -1160.815,E2 -1160.815} C_VEL
LIN {X 0,Y 594.372,Z 448.787,A -85,B 0,C 180,E1 -1161.672,E2 -1161.672} C_VEL
LIN {X 0,Y 594.316,Z 457.69,A -85,B 0,C 180,E1 -1162.697,E2 -1162.697} C_VEL
LIN {X 0,Y 594.281,Z 464.169,A -85,B 0,C 180,E1 -1163.615,E2 -1163.615} C_VEL
LIN {X 0,Y 594.289,Z 469.68,A -85,B 0,C 180,E1 -1164.571,E2 -1164.571} C_VEL
LIN {X 0,Y 594.27,Z 474.371,A -85,B 0,C 180,E1 -1165.591,E2 -1165.591} C_VEL
LIN {X 0,Y 594.267,Z 477.956,A -85,B 0,C 180,E1 -1166.61,E2 -1166.61} C_VEL
LIN {X 0,Y 594.226,Z 479.809,A -85,B 0,C 180,E1 -1167.288,E2 -1167.288} C_VEL
LIN {X 0,Y 594.242,Z 481.201,A -85,B 0,C 180,E1 -1167.967,E2 -1167.967} C_VEL
LIN {X 0,Y 594.239,Z 482.784,A -85,B 0,C 180,E1 -1169.322,E2 -1169.322} C_VEL
LIN {X 0,Y 594.236,Z 483,A -85,B 0,C 180,E1 -1170,E2 -1170} C_VEL
LIN {X 0,Y 594.247,Z 482.185,A -85,B 0,C 180,E1 -1171.355,E2 -1171.355} C_VEL
LIN {X 0,Y 594.242,Z 481.202,A -85,B 0,C 180,E1 -1172.033,E2 -1172.033} C_VEL
LIN {X 0,Y 594.226,Z 479.809,A -85,B 0,C 180,E1 -1172.712,E2 -1172.712} C_VEL
LIN {X 0,Y 594.289,Z 476.896,A -85,B 0,C 180,E1 -1173.729,E2 -1173.729} C_VEL
LIN {X 0,Y 594.241,Z 472.949,A -85,B 0,C 180,E1 -1174.749,E2 -1174.749} C_VEL
LIN {X 0,Y 594.305,Z 466.877,A -85,B 0,C 180,E1 -1175.939,E2 -1175.939} C_VEL
LIN {X 0,Y 594.308,Z 460.235,A -85,B 0,C 180,E1 -1176.962,E2 -1176.962} C_VEL
LIN {X 0,Y 594.359,Z 451.989,A -85,B 0,C 180,E1 -1177.986,E2 -1177.986} C_VEL
LIN {X 0,Y 594.382,Z 443.536,A -85,B 0,C 180,E1 -1178.842,E2 -1178.842} C_VEL
LIN {X 0,Y 594.431,Z 433.092,A -85,B 0,C 180,E1 -1179.699,E2 -1179.699} C_VEL
LIN {X 0,Y 594.459,Z 422.757,A -85,B 0,C 180,E1 -1180.387,E2 -1180.387} C_VEL
LIN {X 0,Y 594.508,Z 410.692,A -85,B 0,C 180,E1 -1181.022,E2 -1181.022} C_VEL
LIN {X 0,Y 594.593,Z 398.477,A -85,B 0,C 180,E1 -1181.505,E2 -1181.505} C_VEL
LIN {X 0,Y 594.652,Z 385.432,A -85,B 0,C 180,E1 -1181.872,E2 -1181.872} C_VEL
LIN {X 0,Y 594.564,Z 376.665,A -85,B 0,C 180,E1 -1182.038,E2 -1182.038} C_VEL
LIN {X 0,Y 594.294,Z 374.976,A -85,B 0,C 180,E1 -1182.074,E2 -1182.074} C_VEL
LIN {X 0,Y 594.32,Z 365.274,A -85,B 0,C 180,E1 -1184.379,E2 -1184.379} C_VEL
LIN {X 0,Y 594.354,Z 353.558,A -85,B 0,C 180,E1 -1187.195,E2 -1187.195} C_VEL
LIN {X 0,Y 594.395,Z 341.843,A -85,B 0,C 180,E1 -1190.053,E2 -1190.053} C_VEL
LIN {X 0,Y 594.403,Z 332.045,A -85,B 0,C 180,E1 -1192.485,E2 -1192.485} C_VEL
LIN {X 0,Y 594.502,Z 321.34,A -85,B 0,C 180,E1 -1195.188,E2 -1195.188} C_VEL
LIN {X 0,Y 594.575,Z 309.531,A -85,B 0,C 180,E1 -1198.217,E2 -1198.217} C_VEL
LIN {X 0,Y 594.525,Z 298.72,A -85,B 0,C 180,E1 -1200.946,E2 -1200.946} C_VEL
LIN {X 0,Y 594.582,Z 288.213,A -85,B 0,C 180,E1 -1203.749,E2 -1203.749} C_VEL
LIN {X 0,Y 594.644,Z 282.294,A -85,B 0,C 180,E1 -1205.389,E2 -1205.389} C_VEL
LIN {X 0,Y 594.378,Z 280.451,A -85,B 0,C 180,E1 -1205.929,E2 -1205.929} C_VEL
LIN {X 0,Y 594.385,Z 280.449,A -85,B 0,C 180,E1 -1208.805,E2 -1208.805} C_VEL
LIN {X 0,Y 594.387,Z 280.449,A -85,B 0,C 180,E1 -1211.848,E2 -1211.848} C_VEL
LIN {X 0,Y 594.369,Z 280.451,A -85,B 0,C 180,E1 -1214.809,E2 -1214.809} C_VEL
LIN {X 0,Y 594.37,Z 280.45,A -85,B 0,C 180,E1 -1217.624,E2 -1217.624} C_VEL
LIN {X 0,Y 594.397,Z 280.447,A -85,B 0,C 180,E1 -1220.321,E2 -1220.321} C_VEL
LIN {X 0,Y 594.388,Z 280.449,A -85,B 0,C 180,E1 -1222.913,E2 -1222.913} C_VEL
LIN {X 0,Y 594.385,Z 280.449,A -85,B 0,C 180,E1 -1225.862,E2 -1225.862} C_VEL
LIN {X 0,Y 594.396,Z 280.447,A -85,B 0,C 180,E1 -1228.651,E2 -1228.651} C_VEL
LIN {X 0,Y 594.388,Z 280.45,A -85,B 0,C 180,E1 -1231.042,E2 -1231.042} C_VEL
LIN {X 0,Y 594.391,Z 280.449,A -85,B 0,C 180,E1 -1233.978,E2 -1233.978} C_VEL
LIN {X 0,Y 594.393,Z 280.448,A -85,B 0,C 180,E1 -1236.296,E2 -1236.296} C_VEL
LIN {X 0,Y 594.405,Z 280.447,A -85,B 0,C 180,E1 -1239.224,E2 -1239.224} C_VEL
LIN {X 0,Y 594.359,Z 280.454,A -85,B 0,C 180,E1 -1242.095,E2 -1242.095} C_VEL
LIN {X 0,Y 594.369,Z 280.451,A -85,B 0,C 180,E1 -1244.219,E2 -1244.219} C_VEL
LIN {X 0,Y 594.387,Z 280.448,A -85,B 0,C 180,E1 -1246.321,E2 -1246.321} C_VEL
LIN {X 0,Y 594.377,Z 280.451,A -85,B 0,C 180,E1 -1249.095,E2 -1249.095} C_VEL
LIN {X 0,Y 594.387,Z 280.448,A -85,B 0,C 180,E1 -1251.843,E2 -1251.843} C_VEL
LIN {X 0,Y 594.391,Z 280.447,A -85,B 0,C 180,E1 -1254.572,E2 -1254.572} C_VEL
LIN {X 0,Y 594.408,Z 280.446,A -85,B 0,C 180,E1 -1257.289,E2 -1257.289} C_VEL
LIN {X 0,Y 594.421,Z 280.445,A -85,B 0,C 180,E1 -1260,E2 -1260} C_VEL
LIN {X 0,Y 594.404,Z 280.446,A -85,B 0,C 180,E1 -1262.711,E2 -1262.711} C_VEL
LIN {X 0,Y 594.399,Z 280.447,A -85,B 0,C 180,E1 -1265.428,E2 -1265.428} C_VEL
LIN {X 0,Y 594.417,Z 280.447,A -85,B 0,C 180,E1 -1268.157,E2 -1268.157} C_VEL
LIN {X 0,Y 594.289,Z 280.463,A -85,B 0,C 180,E1 -1269.53,E2 -1269.53} C_VEL
LIN {X 0,Y 594.252,Z 281.648,A -85,B 0,C 180,E1 -1271.003,E2 -1271.003} C_VEL
LIN {X 0,Y 594.249,Z 284.697,A -85,B 0,C 180,E1 -1273.682,E2 -1273.682} C_VEL
LIN {X 0,Y 594.247,Z 286.582,A -85,B 0,C 180,E1 -1275.267,E2 -1275.267} C_VEL
LIN {X 0,Y 593.563,Z 287.287,A -85,B 0,C 180,E1 -1275.829,E2 -1275.829} C_VEL
LIN {X 0,Y 590.676,Z 288.513,A -85,B 0,C 180,E1 -1276.738,E2 -1276.738} C_VEL
LIN {X 0,Y 588.245,Z 289.501,A -85,B 0,C 180,E1 -1277.47,E2 -1277.47} C_VEL
LIN {X 0,Y 587.204,Z 290.227,A -85,B 0,C 180,E1 -1278.035,E2 -1278.035} C_VEL
LIN {X 0,Y 587.121,Z 290.461,A -85,B 0,C 180,E1 -1278.227,E2 -1278.227} C_VEL
LIN {X 0,Y 587.144,Z 293.887,A -85,B 0,C 180,E1 -1281.045,E2 -1281.045} C_VEL
LIN {X 0,Y 587.11,Z 296.628,A -85,B 0,C 180,E1 -1283.268,E2 -1283.268} C_VEL
LIN {X 0,Y 587.126,Z 299.903,A -85,B 0,C 180,E1 -1285.895,E2 -1285.895} C_VEL
LIN {X 0,Y 587.687,Z 305.486,A -85,B 0,C 180,E1 -1286.032,E2 -1286.032} C_VEL
LIN {X 0,Y 587.651,Z 318.618,A -85,B 0,C 180,E1 -1286.407,E2 -1286.407} C_VEL
LIN {X 0,Y 587.574,Z 330.669,A -85,B 0,C 180,E1 -1286.89,E2 -1286.89} C_VEL
LIN {X 0,Y 587.481,Z 342.549,A -85,B 0,C 180,E1 -1287.521,E2 -1287.521} C_VEL
LIN {X 0,Y 587.437,Z 354.025,A -85,B 0,C 180,E1 -1288.299,E2 -1288.299} C_VEL
LIN {X 0,Y 587.334,Z 363.899,A -85,B 0,C 180,E1 -1289.13,E2 -1289.13} C_VEL
LIN {X 0,Y 587.289,Z 372.1,A -85,B 0,C 180,E1 -1289.975,E2 -1289.975} C_VEL
LIN {X 0,Y 587.254,Z 380.037,A -85,B 0,C 180,E1 -1290.971,E2 -1290.971} C_VEL
LIN {X 0,Y 587.22,Z 386.549,A -85,B 0,C 180,E1 -1291.978,E2 -1291.978} C_VEL
LIN {X 0,Y 587.172,Z 392.261,A -85,B 0,C 180,E1 -1293.086,E2 -1293.086} C_VEL
LIN {X 0,Y 587.159,Z 397.05,A -85,B 0,C 180,E1 -1294.32,E2 -1294.32} C_VEL
LIN {X 0,Y 587.141,Z 400.274,A -85,B 0,C 180,E1 -1295.516,E2 -1295.516} C_VEL
LIN {X 0,Y 587.125,Z 402.288,A -85,B 0,C 180,E1 -1296.763,E2 -1296.763} C_VEL
LIN {X 0,Y 587.121,Z 402.953,A -85,B 0,C 180,E1 -1297.81,E2 -1297.81} C_VEL
LIN {X 0,Y 587.116,Z 402.66,A -85,B 0,C 180,E1 -1298.915,E2 -1298.915} C_VEL
LIN {X 0,Y 587.146,Z 400.911,A -85,B 0,C 180,E1 -1300.268,E2 -1300.268} C_VEL
LIN {X 0,Y 587.167,Z 397.487,A -85,B 0,C 180,E1 -1301.628,E2 -1301.628} C_VEL
LIN {X 0,Y 587.179,Z 394.188,A -85,B 0,C 180,E1 -1302.552,E2 -1302.552} C_VEL
LIN {X 0,Y 587.183,Z 388.651,A -85,B 0,C 180,E1 -1303.735,E2 -1303.735} C_VEL
LIN {X 0,Y 587.219,Z 381.455,A -85,B 0,C 180,E1 -1304.921,E2 -1304.921} C_VEL
LIN {X 0,Y 587.266,Z 374.016,A -85,B 0,C 180,E1 -1305.893,E2 -1305.893} C_VEL
LIN {X 0,Y 587.349,Z 364.743,A -85,B 0,C 180,E1 -1306.878,E2 -1306.878} C_VEL
LIN {X 0,Y 587.425,Z 355.208,A -85,B 0,C 180,E1 -1307.703,E2 -1307.703} C_VEL
LIN {X 0,Y 587.446,Z 345.385,A -85,B 0,C 180,E1 -1308.395,E2 -1308.395} C_VEL
LIN {X 0,Y 587.518,Z 334.221,A -85,B 0,C 180,E1 -1309.027,E2 -1309.027} C_VEL
LIN {X 0,Y 587.645,Z 322.359,A -85,B 0,C 180,E1 -1309.548,E2 -1309.548} C_VEL
LIN {X 0,Y 587.676,Z 309.749,A -85,B 0,C 180,E1 -1309.955,E2 -1309.955} C_VEL
LIN {X 0,Y 587.486,Z 302.267,A -85,B 0,C 180,E1 -1310.131,E2 -1310.131} C_VEL
LIN {X 0,Y 587.144,Z 299.904,A -85,B 0,C 180,E1 -1310.194,E2 -1310.194} C_VEL
LIN {X 0,Y 587.124,Z 296.01,A -85,B 0,C 180,E1 -1313.322,E2 -1313.322} C_VEL
LIN {X 0,Y 587.135,Z 293.007,A -85,B 0,C 180,E1 -1315.765,E2 -1315.765} C_VEL
LIN {X 0,Y 587.149,Z 290.031,A -85,B 0,C 180,E1 -1318.219,E2 -1318.219} C_VEL
LIN {X 0,Y 587.157,Z 286.833,A -85,B 0,C 180,E1 -1320.9,E2 -1320.9} C_VEL
LIN {X 0,Y 587.162,Z 283.594,A -85,B 0,C 180,E1 -1323.713,E2 -1323.713} C_VEL
LIN {X 0,Y 587.183,Z 281.347,A -85,B 0,C 180,E1 -1325.987,E2 -1325.987} C_VEL
LIN {X 0,Y 587.314,Z 281.331,A -85,B 0,C 180,E1 -1328.225,E2 -1328.225} C_VEL
LIN {X 0,Y 587.342,Z 281.325,A -85,B 0,C 180,E1 -1331.151,E2 -1331.151} C_VEL
LIN {X 0,Y 587.328,Z 281.325,A -85,B 0,C 180,E1 -1334.025,E2 -1334.025} C_VEL
LIN {X 0,Y 587.316,Z 281.327,A -85,B 0,C 180,E1 -1336.858,E2 -1336.858} C_VEL
LIN {X 0,Y 587.338,Z 281.325,A -85,B 0,C 180,E1 -1339.66,E2 -1339.66} C_VEL
LIN {X 0,Y 587.369,Z 281.322,A -85,B 0,C 180,E1 -1342.437,E2 -1342.437} C_VEL
LIN {X 0,Y 587.363,Z 281.324,A -85,B 0,C 180,E1 -1345.195,E2 -1345.195} C_VEL
LIN {X 0,Y 587.373,Z 281.324,A -85,B 0,C 180,E1 -1347.943,E2 -1347.943} C_VEL
LIN {X 0,Y 587.391,Z 281.32,A -85,B 0,C 180,E1 -1350.686,E2 -1350.686} C_VEL
LIN {X 0,Y 587.34,Z 281.325,A -85,B 0,C 180,E1 -1353.43,E2 -1353.43} C_VEL
LIN {X 0,Y 587.346,Z 281.324,A -85,B 0,C 180,E1 -1355.493,E2 -1355.493} C_VEL
LIN {X 0,Y 587.366,Z 281.323,A -85,B 0,C 180,E1 -1358.255,E2 -1358.255} C_VEL
LIN {X 0,Y 587.351,Z 281.326,A -85,B 0,C 180,E1 -1361.134,E2 -1361.134} C_VEL
LIN {X 0,Y 587.346,Z 281.325,A -85,B 0,C 180,E1 -1363.846,E2 -1363.846} C_VEL
LIN {X 0,Y 587.344,Z 281.323,A -85,B 0,C 180,E1 -1366.812,E2 -1366.812} C_VEL
LIN {X 0,Y 587.315,Z 281.326,A -85,B 0,C 180,E1 -1369.576,E2 -1369.576} C_VEL
LIN {X 0,Y 587.338,Z 281.325,A -85,B 0,C 180,E1 -1372.514,E2 -1372.514} C_VEL
LIN {X 0,Y 587.352,Z 281.322,A -85,B 0,C 180,E1 -1374.759,E2 -1374.759} C_VEL
LIN {X 0,Y 587.347,Z 281.324,A -85,B 0,C 180,E1 -1377.818,E2 -1377.818} C_VEL
LIN {X 0,Y 587.329,Z 281.327,A -85,B 0,C 180,E1 -1380.508,E2 -1380.508} C_VEL
LIN {X 0,Y 587.337,Z 281.326,A -85,B 0,C 180,E1 -1383.111,E2 -1383.111} C_VEL
LIN {X 0,Y 587.294,Z 281.333,A -85,B 0,C 180,E1 -1385.9,E2 -1385.9} C_VEL
LIN {X 0,Y 587.325,Z 281.329,A -85,B 0,C 180,E1 -1388.48,E2 -1388.48} C_VEL
LIN {X 0,Y 587.336,Z 281.328,A -85,B 0,C 180,E1 -1391.157,E2 -1391.157} C_VEL
LIN {X 0,Y 587.315,Z 281.328,A -85,B 0,C 180,E1 -1394.112,E2 -1394.112} C_VEL
LIN {X 0,Y 587.318,Z 281.326,A -85,B 0,C 180,E1 -1396.994,E2 -1396.994} C_VEL
LIN {X 0,Y 587.316,Z 281.327,A -85,B 0,C 180,E1 -1399.746,E2 -1399.746} C_VEL
LIN {X 0,Y 587.349,Z 281.322,A -85,B 0,C 180,E1 -1402.393,E2 -1402.393} C_VEL
LIN {X 0,Y 587.344,Z 281.327,A -85,B 0,C 180,E1 -1405.654,E2 -1405.654} C_VEL
LIN {X 0,Y 587.339,Z 281.327,A -85,B 0,C 180,E1 -1408.231,E2 -1408.231} C_VEL
LIN {X 0,Y 587.347,Z 281.326,A -85,B 0,C 180,E1 -1410.868,E2 -1410.868} C_VEL
LIN {X 0,Y 587.343,Z 281.324,A -85,B 0,C 180,E1 -1413.823,E2 -1413.823} C_VEL
LIN {X 0,Y 587.306,Z 281.33,A -85,B 0,C 180,E1 -1415.992,E2 -1415.992} C_VEL
LIN {X 0,Y 587.327,Z 281.325,A -85,B 0,C 180,E1 -1418.226,E2 -1418.226} C_VEL
LIN {X 0,Y 587.355,Z 281.323,A -85,B 0,C 180,E1 -1421.151,E2 -1421.151} C_VEL
LIN {X 0,Y 587.312,Z 281.331,A -85,B 0,C 180,E1 -1424.025,E2 -1424.025} C_VEL
LIN {X 0,Y 587.362,Z 281.321,A -85,B 0,C 180,E1 -1426.154,E2 -1426.154} C_VEL
LIN {X 0,Y 587.346,Z 281.324,A -85,B 0,C 180,E1 -1428.963,E2 -1428.963} C_VEL
LIN {X 0,Y 587.345,Z 281.326,A -85,B 0,C 180,E1 -1431.745,E2 -1431.745} C_VEL
LIN {X 0,Y 587.358,Z 281.325,A -85,B 0,C 180,E1 -1434.507,E2 -1434.507} C_VEL
LIN {X 0,Y 587.375,Z 281.323,A -85,B 0,C 180,E1 -1437.257,E2 -1437.257} C_VEL
LIN {X 0,Y 587.388,Z 281.32,A -85,B 0,C 180,E1 -1440,E2 -1440} C_VEL
LIN {X 0,Y 587.366,Z 281.322,A -85,B 0,C 180,E1 -1442.743,E2 -1442.743} C_VEL
LIN {X 0,Y 587.362,Z 281.321,A -85,B 0,C 180,E1 -1445.493,E2 -1445.493} C_VEL
LIN {X 0,Y 587.346,Z 281.323,A -85,B 0,C 180,E1 -1448.256,E2 -1448.256} C_VEL
LIN {X 0,Y 587.355,Z 281.322,A -85,B 0,C 180,E1 -1451.134,E2 -1451.134} C_VEL
LIN {X 0,Y 587.347,Z 281.327,A -85,B 0,C 180,E1 -1454.251,E2 -1454.251} C_VEL
LIN {X 0,Y 587.346,Z 281.323,A -85,B 0,C 180,E1 -1457.406,E2 -1457.406} C_VEL
LIN {X 0,Y 587.325,Z 281.326,A -85,B 0,C 180,E1 -1460.305,E2 -1460.305} C_VEL
LIN {X 0,Y 587.311,Z 281.33,A -85,B 0,C 180,E1 -1463.259,E2 -1463.259} C_VEL
LIN {X 0,Y 587.334,Z 281.324,A -85,B 0,C 180,E1 -1465.517,E2 -1465.517} C_VEL
LIN {X 0,Y 587.31,Z 281.328,A -85,B 0,C 180,E1 -1467.82,E2 -1467.82} C_VEL
LIN {X 0,Y 587.326,Z 281.325,A -85,B 0,C 180,E1 -1470.507,E2 -1470.507} C_VEL
LIN {X 0,Y 587.339,Z 281.323,A -85,B 0,C 180,E1 -1473.397,E2 -1473.397} C_VEL
LIN {X 0,Y 587.285,Z 281.33,A -85,B 0,C 180,E1 -1475.901,E2 -1475.901} C_VEL
LIN {X 0,Y 587.324,Z 281.326,A -85,B 0,C 180,E1 -1478.48,E2 -1478.48} C_VEL
LIN {X 0,Y 587.34,Z 281.323,A -85,B 0,C 180,E1 -1481.157,E2 -1481.157} C_VEL
LIN {X 0,Y 587.316,Z 281.328,A -85,B 0,C 180,E1 -1484.112,E2 -1484.112} C_VEL
LIN {X 0,Y 587.304,Z 281.332,A -85,B 0,C 180,E1 -1486.992,E2 -1486.992} C_VEL
LIN {X 0,Y 587.315,Z 281.331,A -85,B 0,C 180,E1 -1489.745,E2 -1489.745} C_VEL
LIN {X 0,Y 587.346,Z 281.327,A -85,B 0,C 180,E1 -1492.392,E2 -1492.392} C_VEL
LIN {X 0,Y 587.352,Z 281.436,A -85,B 0,C 180,E1 -1493.786,E2 -1493.786} C_VEL
LIN {X 0,Y 587.71,Z 285.5,A -85,B 0,C 180,E1 -1494.97,E2 -1494.97} C_VEL
LIN {X 0,Y 587.667,Z 295.746,A -85,B 0,C 180,E1 -1497.82,E2 -1497.82} C_VEL
LIN {X 0,Y 587.561,Z 307.042,A -85,B 0,C 180,E1 -1500.83,E2 -1500.83} C_VEL
LIN {X 0,Y 587.529,Z 316.919,A -85,B 0,C 180,E1 -1503.348,E2 -1503.348} C_VEL
LIN {X 0,Y 587.451,Z 327.198,A -85,B 0,C 180,E1 -1505.998,E2 -1505.998} C_VEL
LIN {X 0,Y 587.372,Z 338.914,A -85,B 0,C 180,E1 -1508.964,E2 -1508.964} C_VEL
LIN {X 0,Y 587.342,Z 349.165,A -85,B 0,C 180,E1 -1511.513,E2 -1511.513} C_VEL
LIN {X 0,Y 587.298,Z 360.881,A -85,B 0,C 180,E1 -1514.38,E2 -1514.38} C_VEL
LIN {X 0,Y 587.244,Z 372.597,A -85,B 0,C 180,E1 -1517.208,E2 -1517.208} C_VEL
LIN {X 0,Y 587.228,Z 374.976,A -85,B 0,C 180,E1 -1517.779,E2 -1517.779} C_VEL
LIN {X 0,Y 587.74,Z 380.083,A -85,B 0,C 180,E1 -1517.877,E2 -1517.877} C_VEL
LIN {X 0,Y 587.665,Z 393.734,A -85,B 0,C 180,E1 -1518.204,E2 -1518.204} C_VEL
LIN {X 0,Y 587.577,Z 406.333,A -85,B 0,C 180,E1 -1518.653,E2 -1518.653} C_VEL
LIN {X 0,Y 587.498,Z 418.209,A -85,B 0,C 180,E1 -1519.227,E2 -1519.227} C_VEL
LIN {X 0,Y 587.464,Z 429.477,A -85,B 0,C 180,E1 -1519.923,E2 -1519.923} C_VEL
LIN {X 0,Y 587.384,Z 439.646,A -85,B 0,C 180,E1 -1520.704,E2 -1520.704} C_VEL
LIN {X 0,Y 587.34,Z 448.786,A -85,B 0,C 180,E1 -1521.571,E2 -1521.571} C_VEL
LIN {X 0,Y 587.259,Z 457.69,A -85,B 0,C 180,E1 -1522.608,E2 -1522.608} C_VEL
LIN {X 0,Y 587.195,Z 464.745,A -85,B 0,C 180,E1 -1523.627,E2 -1523.627} C_VEL
LIN {X 0,Y 587.211,Z 469.68,A -85,B 0,C 180,E1 -1524.506,E2 -1524.506} C_VEL
LIN {X 0,Y 587.188,Z 474.371,A -85,B 0,C 180,E1 -1525.538,E2 -1525.538} C_VEL
LIN {X 0,Y 587.193,Z 477.956,A -85,B 0,C 180,E1 -1526.569,E2 -1526.569} C_VEL
LIN {X 0,Y 587.132,Z 479.809,A -85,B 0,C 180,E1 -1527.256,E2 -1527.256} C_VEL
LIN {X 0,Y 587.141,Z 481.2,A -85,B 0,C 180,E1 -1527.942,E2 -1527.942} C_VEL
LIN {X 0,Y 587.14,Z 482.784,A -85,B 0,C 180,E1 -1529.314,E2 -1529.314} C_VEL
LIN {X 0,Y 587.137,Z 483,A -85,B 0,C 180,E1 -1530,E2 -1530} C_VEL
LIN {X 0,Y 587.147,Z 482.185,A -85,B 0,C 180,E1 -1531.372,E2 -1531.372} C_VEL
LIN {X 0,Y 587.141,Z 481.201,A -85,B 0,C 180,E1 -1532.058,E2 -1532.058} C_VEL
LIN {X 0,Y 587.132,Z 479.81,A -85,B 0,C 180,E1 -1532.744,E2 -1532.744} C_VEL
LIN {X 0,Y 587.213,Z 476.896,A -85,B 0,C 180,E1 -1533.774,E2 -1533.774} C_VEL
LIN {X 0,Y 587.147,Z 472.949,A -85,B 0,C 180,E1 -1534.806,E2 -1534.806} C_VEL
LIN {X 0,Y 587.218,Z 466.877,A -85,B 0,C 180,E1 -1536.011,E2 -1536.011} C_VEL
LIN {X 0,Y 587.245,Z 460.236,A -85,B 0,C 180,E1 -1537.046,E2 -1537.046} C_VEL
LIN {X 0,Y 587.299,Z 451.989,A -85,B 0,C 180,E1 -1538.083,E2 -1538.083} C_VEL
LIN {X 0,Y 587.343,Z 443.537,A -85,B 0,C 180,E1 -1538.949,E2 -1538.949} C_VEL
LIN {X 0,Y 587.416,Z 433.094,A -85,B 0,C 180,E1 -1539.816,E2 -1539.816} C_VEL
LIN {X 0,Y 587.478,Z 422.756,A -85,B 0,C 180,E1 -1540.512,E2 -1540.512} C_VEL
LIN {X 0,Y 587.533,Z 411.131,A -85,B 0,C 180,E1 -1541.135,E2 -1541.135} C_VEL
LIN {X 0,Y 587.627,Z 398.675,A -85,B 0,C 180,E1 -1541.637,E2 -1541.637} C_VEL
LIN {X 0,Y 587.717,Z 385.431,A -85,B 0,C 180,E1 -1542.014,E2 -1542.014} C_VEL
LIN {X 0,Y 587.544,Z 377.144,A -85,B 0,C 180,E1 -1542.177,E2 -1542.177} C_VEL
LIN {X 0,Y 587.229,Z 374.976,A -85,B 0,C 180,E1 -1542.221,E2 -1542.221} C_VEL
LIN {X 0,Y 587.279,Z 363.81,A -85,B 0,C 180,E1 -1544.91,E2 -1544.91} C_VEL
LIN {X 0,Y 587.325,Z 352.094,A -85,B 0,C 180,E1 -1547.767,E2 -1547.767} C_VEL
LIN {X 0,Y 587.353,Z 341.843,A -85,B 0,C 180,E1 -1550.304,E2 -1550.304} C_VEL
LIN {X 0,Y 587.381,Z 333.056,A -85,B 0,C 180,E1 -1552.512,E2 -1552.512} C_VEL
LIN {X 0,Y 587.498,Z 322.805,A -85,B 0,C 180,E1 -1555.13,E2 -1555.13} C_VEL
LIN {X 0,Y 587.56,Z 312.253,A -85,B 0,C 180,E1 -1557.807,E2 -1557.807} C_VEL
LIN {X 0,Y 587.534,Z 301.496,A -85,B 0,C 180,E1 -1560.542,E2 -1560.542} C_VEL
LIN {X 0,Y 587.612,Z 290.969,A -85,B 0,C 180,E1 -1563.379,E2 -1563.379} C_VEL
LIN {X 0,Y 587.611,Z 283.151,A -85,B 0,C 180,E1 -1565.58,E2 -1565.58} C_VEL
LIN {X 0,Y 587.333,Z 281.329,A -85,B 0,C 180,E1 -1566.162,E2 -1566.162} C_VEL
LIN {X 0,Y 587.33,Z 281.329,A -85,B 0,C 180,E1 -1568.941,E2 -1568.941} C_VEL
LIN {X 0,Y 587.34,Z 281.327,A -85,B 0,C 180,E1 -1571.157,E2 -1571.157} C_VEL
LIN {X 0,Y 587.332,Z 281.329,A -85,B 0,C 180,E1 -1574.114,E2 -1574.114} C_VEL
LIN {X 0,Y 587.318,Z 281.331,A -85,B 0,C 180,E1 -1576.994,E2 -1576.994} C_VEL
LIN {X 0,Y 587.321,Z 281.329,A -85,B 0,C 180,E1 -1579.746,E2 -1579.746} C_VEL
LIN {X 0,Y 587.35,Z 281.325,A -85,B 0,C 180,E1 -1582.393,E2 -1582.393} C_VEL
LIN {X 0,Y 587.366,Z 281.323,A -85,B 0,C 180,E1 -1585.78,E2 -1585.78} C_VEL
LIN {X 0,Y 587.354,Z 281.325,A -85,B 0,C 180,E1 -1588.232,E2 -1588.232} C_VEL
LIN {X 0,Y 587.355,Z 281.324,A -85,B 0,C 180,E1 -1590.867,E2 -1590.867} C_VEL
LIN {X 0,Y 587.365,Z 281.323,A -85,B 0,C 180,E1 -1593.819,E2 -1593.819} C_VEL
LIN {X 0,Y 587.341,Z 281.327,A -85,B 0,C 180,E1 -1595.994,E2 -1595.994} C_VEL
LIN {X 0,Y 587.324,Z 281.329,A -85,B 0,C 180,E1 -1598.226,E2 -1598.226} C_VEL
LIN {X 0,Y 587.353,Z 281.326,A -85,B 0,C 180,E1 -1601.151,E2 -1601.151} C_VEL
LIN {X 0,Y 587.323,Z 281.329,A -85,B 0,C 180,E1 -1604.025,E2 -1604.025} C_VEL
LIN {X 0,Y 587.365,Z 281.324,A -85,B 0,C 180,E1 -1606.154,E2 -1606.154} C_VEL
LIN {X 0,Y 587.344,Z 281.326,A -85,B 0,C 180,E1 -1608.962,E2 -1608.962} C_VEL
LIN {X 0,Y 587.347,Z 281.325,A -85,B 0,C 180,E1 -1611.744,E2 -1611.744} C_VEL
LIN {X 0,Y 587.357,Z 281.324,A -85,B 0,C 180,E1 -1614.507,E2 -1614.507} C_VEL
LIN {X 0,Y 587.375,Z 281.323,A -85,B 0,C 180,E1 -1617.257,E2 -1617.257} C_VEL
LIN {X 0,Y 587.39,Z 281.321,A -85,B 0,C 180,E1 -1620,E2 -1620} C_VEL
LIN {X 0,Y 587.372,Z 281.322,A -85,B 0,C 180,E1 -1622.743,E2 -1622.743} C_VEL
LIN {X 0,Y 587.364,Z 281.323,A -85,B 0,C 180,E1 -1625.493,E2 -1625.493} C_VEL
LIN {X 0,Y 587.367,Z 281.324,A -85,B 0,C 180,E1 -1628.255,E2 -1628.255} C_VEL
LIN {X 0,Y 587.225,Z 281.343,A -85,B 0,C 180,E1 -1629.646,E2 -1629.646} C_VEL
LIN {X 0,Y 587.203,Z 282.339,A -85,B 0,C 180,E1 -1631.058,E2 -1631.058} C_VEL
LIN {X 0,Y 587.177,Z 285.258,A -85,B 0,C 180,E1 -1633.85,E2 -1633.85} C_VEL
LIN {X 0,Y 587.149,Z 288.684,A -85,B 0,C 180,E1 -1636.747,E2 -1636.747} C_VEL
LIN {X 0,Y 587.121,Z 290.461,A -85,B 0,C 180,E1 -1638.227,E2 -1638.227} C_VEL
LIN {X 0,Y 586.452,Z 291.175,A -85,B 0,C 180,E1 -1638.795,E2 -1638.795} C_VEL
LIN {X 0,Y 583.579,Z 292.405,A -85,B 0,C 180,E1 -1639.716,E2 -1639.716} C_VEL
LIN {X 0,Y 581.156,Z 293.394,A -85,B 0,C 180,E1 -1640.457,E2 -1640.457} C_VEL
LIN {X 0,Y 580.125,Z 294.125,A -85,B 0,C 180,E1 -1641.029,E2 -1641.029} C_VEL
LIN {X 0,Y 580.047,Z 294.363,A -85,B 0,C 180,E1 -1641.223,E2 -1641.223} C_VEL
LIN {X 0,Y 580.017,Z 297.224,A -85,B 0,C 180,E1 -1643.569,E2 -1643.569} C_VEL
LIN {X 0,Y 580.022,Z 299.9,A -85,B 0,C 180,E1 -1645.741,E2 -1645.741} C_VEL
LIN {X 0,Y 580.738,Z 305.978,A -85,B 0,C 180,E1 -1645.898,E2 -1645.898} C_VEL
LIN {X 0,Y 580.691,Z 319.285,A -85,B 0,C 180,E1 -1646.288,E2 -1646.288} C_VEL
LIN {X 0,Y 580.6,Z 331.655,A -85,B 0,C 180,E1 -1646.801,E2 -1646.801} C_VEL
LIN {X 0,Y 580.489,Z 343.756,A -85,B 0,C 180,E1 -1647.467,E2 -1647.467} C_VEL
LIN {X 0,Y 580.397,Z 354.042,A -85,B 0,C 180,E1 -1648.18,E2 -1648.18} C_VEL
LIN {X 0,Y 580.31,Z 363.413,A -85,B 0,C 180,E1 -1648.975,E2 -1648.975} C_VEL
LIN {X 0,Y 580.23,Z 372.952,A -85,B 0,C 180,E1 -1649.976,E2 -1649.976} C_VEL
LIN {X 0,Y 580.187,Z 380.887,A -85,B 0,C 180,E1 -1651.005,E2 -1651.005} C_VEL
LIN {X 0,Y 580.153,Z 387.142,A -85,B 0,C 180,E1 -1652.006,E2 -1652.006} C_VEL
LIN {X 0,Y 580.096,Z 392.317,A -85,B 0,C 180,E1 -1653.037,E2 -1653.037} C_VEL
LIN {X 0,Y 580.082,Z 396.809,A -85,B 0,C 180,E1 -1654.197,E2 -1654.197} C_VEL
LIN {X 0,Y 580.046,Z 399.48,A -85,B 0,C 180,E1 -1655.136,E2 -1655.136} C_VEL
LIN {X 0,Y 580.017,Z 401.917,A -85,B 0,C 180,E1 -1656.422,E2 -1656.422} C_VEL
LIN {X 0,Y 580.029,Z 402.743,A -85,B 0,C 180,E1 -1657.289,E2 -1657.289} C_VEL
LIN {X 0,Y 580.018,Z 402.979,A -85,B 0,C 180,E1 -1658.167,E2 -1658.167} C_VEL
LIN {X 0,Y 580.022,Z 402.497,A -85,B 0,C 180,E1 -1659.151,E2 -1659.151} C_VEL
LIN {X 0,Y 580.046,Z 401.013,A -85,B 0,C 180,E1 -1660.241,E2 -1660.241} C_VEL
LIN {X 0,Y 580.072,Z 398.575,A -85,B 0,C 180,E1 -1661.307,E2 -1661.307} C_VEL
LIN {X 0,Y 580.081,Z 395.195,A -85,B 0,C 180,E1 -1662.349,E2 -1662.349} C_VEL
LIN {X 0,Y 580.109,Z 390.836,A -85,B 0,C 180,E1 -1663.372,E2 -1663.372} C_VEL
LIN {X 0,Y 580.157,Z 385.435,A -85,B 0,C 180,E1 -1664.379,E2 -1664.379} C_VEL
LIN {X 0,Y 580.172,Z 378.917,A -85,B 0,C 180,E1 -1665.364,E2 -1665.364} C_VEL
LIN {X 0,Y 580.229,Z 371.021,A -85,B 0,C 180,E1 -1666.337,E2 -1666.337} C_VEL
LIN {X 0,Y 580.302,Z 361.421,A -85,B 0,C 180,E1 -1667.295,E2 -1667.295} C_VEL
LIN {X 0,Y 580.436,Z 350.595,A -85,B 0,C 180,E1 -1668.168,E2 -1668.168} C_VEL
LIN {X 0,Y 580.522,Z 338.799,A -85,B 0,C 180,E1 -1668.916,E2 -1668.916} C_VEL
LIN {X 0,Y 580.63,Z 326.096,A -85,B 0,C 180,E1 -1669.54,E2 -1669.54} C_VEL
LIN {X 0,Y 580.72,Z 313.435,A -85,B 0,C 180,E1 -1669.993,E2 -1669.993} C_VEL
LIN {X 0,Y 580.608,Z 303.485,A -85,B 0,C 180,E1 -1670.253,E2 -1670.253} C_VEL
LIN {X 0,Y 580.053,Z 299.909,A -85,B 0,C 180,E1 -1670.341,E2 -1670.341} C_VEL
LIN {X 0,Y 580.031,Z 296.513,A -85,B 0,C 180,E1 -1673.101,E2 -1673.101} C_VEL
LIN {X 0,Y 580.048,Z 293.624,A -85,B 0,C 180,E1 -1675.478,E2 -1675.478} C_VEL
LIN {X 0,Y 580.043,Z 290.586,A -85,B 0,C 180,E1 -1678.01,E2 -1678.01} C_VEL
LIN {X 0,Y 580.084,Z 287.047,A -85,B 0,C 180,E1 -1681.012,E2 -1681.012} C_VEL
LIN {X 0,Y 580.097,Z 284.101,A -85,B 0,C 180,E1 -1683.705,E2 -1683.705} C_VEL
LIN {X 0,Y 580.117,Z 282.227,A -85,B 0,C 180,E1 -1685.675,E2 -1685.675} C_VEL
LIN {X 0,Y 580.255,Z 282.208,A -85,B 0,C 180,E1 -1687.946,E2 -1687.946} C_VEL
LIN {X 0,Y 580.299,Z 282.205,A -85,B 0,C 180,E1 -1690.913,E2 -1690.913} C_VEL
LIN {X 0,Y 580.281,Z 282.203,A -85,B 0,C 180,E1 -1693.825,E2 -1693.825} C_VEL
LIN {X 0,Y 580.273,Z 282.204,A -85,B 0,C 180,E1 -1696.696,E2 -1696.696} C_VEL
LIN {X 0,Y 580.307,Z 282.203,A -85,B 0,C 180,E1 -1698.827,E2 -1698.827} C_VEL
LIN {X 0,Y 580.331,Z 282.198,A -85,B 0,C 180,E1 -1701.644,E2 -1701.644} C_VEL
LIN {X 0,Y 580.315,Z 282.199,A -85,B 0,C 180,E1 -1704.44,E2 -1704.44} C_VEL
LIN {X 0,Y 580.329,Z 282.197,A -85,B 0,C 180,E1 -1707.223,E2 -1707.223} C_VEL
LIN {X 0,Y 580.356,Z 282.193,A -85,B 0,C 180,E1 -1710,E2 -1710} C_VEL
LIN {X 0,Y 580.333,Z 282.197,A -85,B 0,C 180,E1 -1712.777,E2 -1712.777} C_VEL
LIN {X 0,Y 580.313,Z 282.201,A -85,B 0,C 180,E1 -1715.56,E2 -1715.56} C_VEL
LIN {X 0,Y 580.328,Z 282.2,A -85,B 0,C 180,E1 -1718.356,E2 -1718.356} C_VEL
LIN {X 0,Y 580.302,Z 282.203,A -85,B 0,C 180,E1 -1721.191,E2 -1721.191} C_VEL
LIN {X 0,Y 580.306,Z 282.201,A -85,B 0,C 180,E1 -1724.018,E2 -1724.018} C_VEL
LIN {X 0,Y 580.315,Z 282.199,A -85,B 0,C 180,E1 -1726.914,E2 -1726.914} C_VEL
LIN {X 0,Y 580.289,Z 282.202,A -85,B 0,C 180,E1 -1729.823,E2 -1729.823} C_VEL
LIN {X 0,Y 580.267,Z 282.205,A -85,B 0,C 180,E1 -1732.053,E2 -1732.053} C_VEL
LIN {X 0,Y 580.306,Z 282.2,A -85,B 0,C 180,E1 -1735.08,E2 -1735.08} C_VEL
LIN {X 0,Y 580.297,Z 282.204,A -85,B 0,C 180,E1 -1738.186,E2 -1738.186} C_VEL
LIN {X 0,Y 580.283,Z 282.207,A -85,B 0,C 180,E1 -1740.694,E2 -1740.694} C_VEL
LIN {X 0,Y 580.284,Z 282.206,A -85,B 0,C 180,E1 -1743.313,E2 -1743.313} C_VEL
LIN {X 0,Y 580.249,Z 282.209,A -85,B 0,C 180,E1 -1745.757,E2 -1745.757} C_VEL
LIN {X 0,Y 580.286,Z 282.203,A -85,B 0,C 180,E1 -1748.147,E2 -1748.147} C_VEL
LIN {X 0,Y 580.3,Z 282.201,A -85,B 0,C 180,E1 -1750.844,E2 -1750.844} C_VEL
LIN {X 0,Y 580.276,Z 282.206,A -85,B 0,C 180,E1 -1753.659,E2 -1753.659} C_VEL
LIN {X 0,Y 580.278,Z 282.206,A -85,B 0,C 180,E1 -1756.61,E2 -1756.61} C_VEL
LIN {X 0,Y 580.3,Z 282.205,A -85,B 0,C 180,E1 -1759.157,E2 -1759.157} C_VEL
LIN {X 0,Y 580.294,Z 282.203,A -85,B 0,C 180,E1 -1761.927,E2 -1761.927} C_VEL
LIN {X 0,Y 580.256,Z 282.209,A -85,B 0,C 180,E1 -1764.453,E2 -1764.453} C_VEL
LIN {X 0,Y 580.289,Z 282.206,A -85,B 0,C 180,E1 -1766.975,E2 -1766.975} C_VEL
LIN {X 0,Y 580.299,Z 282.203,A -85,B 0,C 180,E1 -1769.425,E2 -1769.425} C_VEL
LIN {X 0,Y 580.292,Z 282.205,A -85,B 0,C 180,E1 -1772.144,E2 -1772.144} C_VEL
LIN {X 0,Y 580.291,Z 282.206,A -85,B 0,C 180,E1 -1774.92,E2 -1774.92} C_VEL
LIN {X 0,Y 580.277,Z 282.203,A -85,B 0,C 180,E1 -1777.948,E2 -1777.948} C_VEL
LIN {X 0,Y 580.304,Z 282.2,A -85,B 0,C 180,E1 -1780.914,E2 -1780.914} C_VEL
LIN {X 0,Y 580.263,Z 282.207,A -85,B 0,C 180,E1 -1783.825,E2 -1783.825} C_VEL
LIN {X 0,Y 580.33,Z 282.196,A -85,B 0,C 180,E1 -1785.983,E2 -1785.983} C_VEL
LIN {X 0,Y 580.311,Z 282.199,A -85,B 0,C 180,E1 -1788.827,E2 -1788.827} C_VEL
LIN {X 0,Y 580.313,Z 282.201,A -85,B 0,C 180,E1 -1791.644,E2 -1791.644} C_VEL
LIN {X 0,Y 580.289,Z 282.202,A -85,B 0,C 180,E1 -1793.742,E2 -1793.742} C_VEL
LIN {X 0,Y 580.27,Z 282.208,A -85,B 0,C 180,E1 -1795.833,E2 -1795.833} C_VEL
LIN {X 0,Y 580.347,Z 282.194,A -85,B 0,C 180,E1 -1797.918,E2 -1797.918} C_VEL
LIN {X 0,Y 580.359,Z 282.194,A -85,B 0,C 180,E1 -1800.694,E2 -1800.694} C_VEL
LIN {X 0,Y 580.331,Z 282.198,A -85,B 0,C 180,E1 -1802.777,E2 -1802.777} C_VEL
LIN {X 0,Y 580.327,Z 282.197,A -85,B 0,C 180,E1 -1805.56,E2 -1805.56} C_VEL
LIN {X 0,Y 580.315,Z 282.199,A -85,B 0,C 180,E1 -1808.356,E2 -1808.356} C_VEL
LIN {X 0,Y 580.307,Z 282.2,A -85,B 0,C 180,E1 -1811.191,E2 -1811.191} C_VEL
LIN {X 0,Y 580.321,Z 282.199,A -85,B 0,C 180,E1 -1814.017,E2 -1814.017} C_VEL
LIN {X 0,Y 580.319,Z 282.202,A -85,B 0,C 180,E1 -1816.914,E2 -1816.914} C_VEL
LIN {X 0,Y 580.286,Z 282.203,A -85,B 0,C 180,E1 -1819.823,E2 -1819.823} C_VEL
LIN {X 0,Y 580.273,Z 282.207,A -85,B 0,C 180,E1 -1822.053,E2 -1822.053} C_VEL
LIN {X 0,Y 580.31,Z 282.2,A -85,B 0,C 180,E1 -1825.08,E2 -1825.08} C_VEL
LIN {X 0,Y 580.285,Z 282.203,A -85,B 0,C 180,E1 -1828.186,E2 -1828.186} C_VEL
LIN {X 0,Y 580.276,Z 282.203,A -85,B 0,C 180,E1 -1830.692,E2 -1830.692} C_VEL
LIN {X 0,Y 580.308,Z 282.199,A -85,B 0,C 180,E1 -1833.316,E2 -1833.316} C_VEL
LIN {X 0,Y 580.235,Z 282.209,A -85,B 0,C 180,E1 -1835.754,E2 -1835.754} C_VEL
LIN {X 0,Y 580.289,Z 282.203,A -85,B 0,C 180,E1 -1838.147,E2 -1838.147} C_VEL
LIN {X 0,Y 580.301,Z 282.201,A -85,B 0,C 180,E1 -1840.843,E2 -1840.843} C_VEL
LIN {X 0,Y 580.274,Z 282.204,A -85,B 0,C 180,E1 -1843.659,E2 -1843.659} C_VEL
LIN {X 0,Y 580.274,Z 282.204,A -85,B 0,C 180,E1 -1846.61,E2 -1846.61} C_VEL
LIN {X 0,Y 580.302,Z 282.2,A -85,B 0,C 180,E1 -1849.156,E2 -1849.156} C_VEL
LIN {X 0,Y 580.29,Z 282.204,A -85,B 0,C 180,E1 -1851.927,E2 -1851.927} C_VEL
LIN {X 0,Y 580.298,Z 282.253,A -85,B 0,C 180,E1 -1853.551,E2 -1853.551} C_VEL
LIN {X 0,Y 580.739,Z 285.369,A -85,B 0,C 180,E1 -1854.487,E2 -1854.487} C_VEL
LIN {X 0,Y 580.729,Z 292.846,A -85,B 0,C 180,E1 -1856.62,E2 -1856.62} C_VEL
LIN {X 0,Y 580.609,Z 302.399,A -85,B 0,C 180,E1 -1859.252,E2 -1859.252} C_VEL
LIN {X 0,Y 580.548,Z 313.16,A -85,B 0,C 180,E1 -1862.095,E2 -1862.095} C_VEL
LIN {X 0,Y 580.5,Z 324.262,A -85,B 0,C 180,E1 -1864.929,E2 -1864.929} C_VEL
LIN {X 0,Y 580.389,Z 335.985,A -85,B 0,C 180,E1 -1867.952,E2 -1867.952} C_VEL
LIN {X 0,Y 580.305,Z 347.701,A -85,B 0,C 180,E1 -1870.913,E2 -1870.913} C_VEL
LIN {X 0,Y 580.264,Z 357.952,A -85,B 0,C 180,E1 -1873.463,E2 -1873.463} C_VEL
LIN {X 0,Y 580.201,Z 369.668,A -85,B 0,C 180,E1 -1876.337,E2 -1876.337} C_VEL
LIN {X 0,Y 580.157,Z 374.976,A -85,B 0,C 180,E1 -1877.627,E2 -1877.627} C_VEL
LIN {X 0,Y 580.795,Z 380.083,A -85,B 0,C 180,E1 -1877.73,E2 -1877.73} C_VEL
LIN {X 0,Y 580.739,Z 393.735,A -85,B 0,C 180,E1 -1878.061,E2 -1878.061} C_VEL
LIN {X 0,Y 580.624,Z 406.316,A -85,B 0,C 180,E1 -1878.515,E2 -1878.515} C_VEL
LIN {X 0,Y 580.519,Z 418.209,A -85,B 0,C 180,E1 -1879.096,E2 -1879.096} C_VEL
LIN {X 0,Y 580.454,Z 429.479,A -85,B 0,C 180,E1 -1879.8,E2 -1879.8} C_VEL
LIN {X 0,Y 580.352,Z 439.646,A -85,B 0,C 180,E1 -1880.591,E2 -1880.591} C_VEL
LIN {X 0,Y 580.279,Z 448.786,A -85,B 0,C 180,E1 -1881.468,E2 -1881.468} C_VEL
LIN {X 0,Y 580.199,Z 457.69,A -85,B 0,C 180,E1 -1882.518,E2 -1882.518} C_VEL
LIN {X 0,Y 580.12,Z 464.465,A -85,B 0,C 180,E1 -1883.505,E2 -1883.505} C_VEL
LIN {X 0,Y 580.139,Z 469.68,A -85,B 0,C 180,E1 -1884.438,E2 -1884.438} C_VEL
LIN {X 0,Y 580.108,Z 474.372,A -85,B 0,C 180,E1 -1885.483,E2 -1885.483} C_VEL
LIN {X 0,Y 580.123,Z 477.957,A -85,B 0,C 180,E1 -1886.527,E2 -1886.527} C_VEL
LIN {X 0,Y 580.043,Z 479.808,A -85,B 0,C 180,E1 -1887.222,E2 -1887.222} C_VEL
LIN {X 0,Y 580.04,Z 481.199,A -85,B 0,C 180,E1 -1887.917,E2 -1887.917} C_VEL
LIN {X 0,Y 580.04,Z 482.785,A -85,B 0,C 180,E1 -1889.306,E2 -1889.306} C_VEL
LIN {X 0,Y 580.037,Z 483,A -85,B 0,C 180,E1 -1890,E2 -1890} C_VEL
LIN {X 0,Y 580.047,Z 482.186,A -85,B 0,C 180,E1 -1891.389,E2 -1891.389} C_VEL
LIN {X 0,Y 580.04,Z 481.2,A -85,B 0,C 180,E1 -1892.083,E2 -1892.083} C_VEL
LIN {X 0,Y 580.043,Z 479.81,A -85,B 0,C 180,E1 -1892.778,E2 -1892.778} C_VEL
LIN {X 0,Y 580.11,Z 476.896,A -85,B 0,C 180,E1 -1893.821,E2 -1893.821} C_VEL
LIN {X 0,Y 580.053,Z 472.949,A -85,B 0,C 180,E1 -1894.865,E2 -1894.865} C_VEL
LIN {X 0,Y 580.139,Z 466.877,A -85,B 0,C 180,E1 -1896.085,E2 -1896.085} C_VEL
LIN {X 0,Y 580.184,Z 460.237,A -85,B 0,C 180,E1 -1897.132,E2 -1897.132} C_VEL
LIN {X 0,Y 580.25,Z 451.989,A -85,B 0,C 180,E1 -1898.182,E2 -1898.182} C_VEL
LIN {X 0,Y 580.308,Z 443.537,A -85,B 0,C 180,E1 -1899.058,E2 -1899.058} C_VEL
LIN {X 0,Y 580.418,Z 433.095,A -85,B 0,C 180,E1 -1899.936,E2 -1899.936} C_VEL
LIN {X 0,Y 580.492,Z 422.755,A -85,B 0,C 180,E1 -1900.64,E2 -1900.64} C_VEL
LIN {X 0,Y 580.563,Z 411.588,A -85,B 0,C 180,E1 -1901.248,E2 -1901.248} C_VEL
LIN {X 0,Y 580.665,Z 399.764,A -85,B 0,C 180,E1 -1901.741,E2 -1901.741} C_VEL
LIN {X 0,Y 580.791,Z 386.344,A -85,B 0,C 180,E1 -1902.137,E2 -1902.137} C_VEL
LIN {X 0,Y 580.576,Z 377.603,A -85,B 0,C 180,E1 -1902.319,E2 -1902.319} C_VEL
LIN {X 0,Y 580.158,Z 374.976,A -85,B 0,C 180,E1 -1902.373,E2 -1902.373} C_VEL
LIN {X 0,Y 580.234,Z 363.81,A -85,B 0,C 180,E1 -1905.095,E2 -1905.095} C_VEL
LIN {X 0,Y 580.286,Z 352.094,A -85,B 0,C 180,E1 -1907.989,E2 -1907.989} C_VEL
LIN {X 0,Y 580.331,Z 341.843,A -85,B 0,C 180,E1 -1910.561,E2 -1910.561} C_VEL
LIN {X 0,Y 580.397,Z 331.312,A -85,B 0,C 180,E1 -1913.247,E2 -1913.247} C_VEL
LIN {X 0,Y 580.493,Z 321.175,A -85,B 0,C 180,E1 -1915.84,E2 -1915.84} C_VEL
LIN {X 0,Y 580.511,Z 310.302,A -85,B 0,C 180,E1 -1918.569,E2 -1918.569} C_VEL
LIN {X 0,Y 580.572,Z 299.689,A -85,B 0,C 180,E1 -1921.368,E2 -1921.368} C_VEL
LIN {X 0,Y 580.673,Z 290.752,A -85,B 0,C 180,E1 -1923.831,E2 -1923.831} C_VEL
LIN {X 0,Y 580.669,Z 284.845,A -85,B 0,C 180,E1 -1925.518,E2 -1925.518} C_VEL
LIN {X 0,Y 580.282,Z 282.206,A -85,B 0,C 180,E1 -1926.362,E2 -1926.362} C_VEL
LIN {X 0,Y 580.302,Z 282.203,A -85,B 0,C 180,E1 -1929.186,E2 -1929.186} C_VEL
LIN {X 0,Y 580.285,Z 282.205,A -85,B 0,C 180,E1 -1931.769,E2 -1931.769} C_VEL
LIN {X 0,Y 580.272,Z 282.206,A -85,B 0,C 180,E1 -1934.626,E2 -1934.626} C_VEL
LIN {X 0,Y 580.291,Z 282.205,A -85,B 0,C 180,E1 -1937.628,E2 -1937.628} C_VEL
LIN {X 0,Y 580.299,Z 282.205,A -85,B 0,C 180,E1 -1940.067,E2 -1940.067} C_VEL
LIN {X 0,Y 580.304,Z 282.204,A -85,B 0,C 180,E1 -1943.066,E2 -1943.066} C_VEL
LIN {X 0,Y 580.321,Z 282.202,A -85,B 0,C 180,E1 -1946.145,E2 -1946.145} C_VEL
LIN {X 0,Y 580.292,Z 282.203,A -85,B 0,C 180,E1 -1948.615,E2 -1948.615} C_VEL
LIN {X 0,Y 580.297,Z 282.205,A -85,B 0,C 180,E1 -1951.024,E2 -1951.024} C_VEL
LIN {X 0,Y 580.297,Z 282.203,A -85,B 0,C 180,E1 -1953.666,E2 -1953.666} C_VEL
LIN {X 0,Y 580.306,Z 282.201,A -85,B 0,C 180,E1 -1955.684,E2 -1955.684} C_VEL
LIN {X 0,Y 580.275,Z 282.206,A -85,B 0,C 180,E1 -1957.947,E2 -1957.947} C_VEL
LIN {X 0,Y 580.303,Z 282.203,A -85,B 0,C 180,E1 -1960.913,E2 -1960.913} C_VEL
LIN {X 0,Y 580.273,Z 282.206,A -85,B 0,C 180,E1 -1963.825,E2 -1963.825} C_VEL
LIN {X 0,Y 580.332,Z 282.2,A -85,B 0,C 180,E1 -1965.983,E2 -1965.983} C_VEL
LIN {X 0,Y 580.312,Z 282.201,A -85,B 0,C 180,E1 -1968.827,E2 -1968.827} C_VEL
LIN {X 0,Y 580.316,Z 282.2,A -85,B 0,C 180,E1 -1971.644,E2 -1971.644} C_VEL
LIN {X 0,Y 580.323,Z 282.2,A -85,B 0,C 180,E1 -1974.44,E2 -1974.44} C_VEL
LIN {X 0,Y 580.347,Z 282.197,A -85,B 0,C 180,E1 -1977.918,E2 -1977.918} C_VEL
LIN {X 0,Y 580.362,Z 282.194,A -85,B 0,C 180,E1 -1980.694,E2 -1980.694} C_VEL
LIN {X 0,Y 580.291,Z 282.204,A -85,B 0,C 180,E1 -1983.472,E2 -1983.472} C_VEL
LIN {X 0,Y 580.329,Z 282.199,A -85,B 0,C 180,E1 -1985.56,E2 -1985.56} C_VEL
LIN {X 0,Y 580.327,Z 282.2,A -85,B 0,C 180,E1 -1988.356,E2 -1988.356} C_VEL
LIN {X 0,Y 580.125,Z 282.467,A -85,B 0,C 180,E1 -1990.47,E2 -1990.47} C_VEL
LIN {X 0,Y 580.092,Z 285.154,A -85,B 0,C 180,E1 -1993.308,E2 -1993.308} C_VEL
LIN {X 0,Y 580.072,Z 287.492,A -85,B 0,C 180,E1 -1995.459,E2 -1995.459} C_VEL
LIN {X 0,Y 580.025,Z 290.761,A -85,B 0,C 180,E1 -1998.226,E2 -1998.226} C_VEL
LIN {X 0,Y 580.046,Z 294.212,A -85,B 0,C 180,E1 -2001.099,E2 -2001.099} C_VEL
LIN {X 0,Y 580.047,Z 294.363,A -85,B 0,C 180,E1 -2001.223,E2 -2001.223} C_VEL
LIN {X 0,Y 579.382,Z 295.085,A -85,B 0,C 180,E1 -2001.799,E2 -2001.799} C_VEL
LIN {X 0,Y 576.482,Z 296.315,A -85,B 0,C 180,E1 -2002.731,E2 -2002.731} C_VEL
LIN {X 0,Y 574.033,Z 297.305,A -85,B 0,C 180,E1 -2003.481,E2 -2003.481} C_VEL
LIN {X 0,Y 572.993,Z 298.041,A -85,B 0,C 180,E1 -2004.061,E2 -2004.061} C_VEL
LIN {X 0,Y 572.915,Z 298.281,A -85,B 0,C 180,E1 -2004.258,E2 -2004.258} C_VEL
LIN {X 0,Y 572.945,Z 299.91,A -85,B 0,C 180,E1 -2005.595,E2 -2005.595} C_VEL
LIN {X 0,Y 573.821,Z 306.914,A -85,B 0,C 180,E1 -2005.772,E2 -2005.772} C_VEL
LIN {X 0,Y 573.737,Z 319.948,A -85,B 0,C 180,E1 -2006.167,E2 -2006.167} C_VEL
LIN {X 0,Y 573.622,Z 331.384,A -85,B 0,C 180,E1 -2006.649,E2 -2006.649} C_VEL
LIN {X 0,Y 573.474,Z 342.543,A -85,B 0,C 180,E1 -2007.26,E2 -2007.26} C_VEL
LIN {X 0,Y 573.371,Z 353.938,A -85,B 0,C 180,E1 -2008.05,E2 -2008.05} C_VEL
LIN {X 0,Y 573.27,Z 364.444,A -85,B 0,C 180,E1 -2008.963,E2 -2008.963} C_VEL
LIN {X 0,Y 573.178,Z 373.912,A -85,B 0,C 180,E1 -2009.991,E2 -2009.991} C_VEL
LIN {X 0,Y 573.123,Z 381.456,A -85,B 0,C 180,E1 -2010.999,E2 -2010.999} C_VEL
LIN {X 0,Y 573.065,Z 388.567,A -85,B 0,C 180,E1 -2012.198,E2 -2012.198} C_VEL
LIN {X 0,Y 572.996,Z 394.484,A -85,B 0,C 180,E1 -2013.5,E2 -2013.5} C_VEL
LIN {X 0,Y 572.99,Z 398.557,A -85,B 0,C 180,E1 -2014.735,E2 -2014.735} C_VEL
LIN {X 0,Y 572.925,Z 401.417,A -85,B 0,C 180,E1 -2016.073,E2 -2016.073} C_VEL
LIN {X 0,Y 572.929,Z 402.638,A -85,B 0,C 180,E1 -2017.122,E2 -2017.122} C_VEL
LIN {X 0,Y 572.931,Z 402.956,A -85,B 0,C 180,E1 -2018.272,E2 -2018.272} C_VEL
LIN {X 0,Y 572.928,Z 401.978,A -85,B 0,C 180,E1 -2019.633,E2 -2019.633} C_VEL
LIN {X 0,Y 572.95,Z 399.417,A -85,B 0,C 180,E1 -2021.014,E2 -2021.014} C_VEL
LIN {X 0,Y 573.003,Z 396.721,A -85,B 0,C 180,E1 -2021.967,E2 -2021.967} C_VEL
LIN {X 0,Y 573.02,Z 392.95,A -85,B 0,C 180,E1 -2022.97,E2 -2022.97} C_VEL
LIN {X 0,Y 573.062,Z 387.137,A -85,B 0,C 180,E1 -2024.16,E2 -2024.16} C_VEL
LIN {X 0,Y 573.086,Z 379.729,A -85,B 0,C 180,E1 -2025.339,E2 -2025.339} C_VEL
LIN {X 0,Y 573.178,Z 371.911,A -85,B 0,C 180,E1 -2026.338,E2 -2026.338} C_VEL
LIN {X 0,Y 573.275,Z 363.455,A -85,B 0,C 180,E1 -2027.223,E2 -2027.223} C_VEL
LIN {X 0,Y 573.382,Z 352.699,A -85,B 0,C 180,E1 -2028.134,E2 -2028.134} C_VEL
LIN {X 0,Y 573.469,Z 341.258,A -85,B 0,C 180,E1 -2028.91,E2 -2028.91} C_VEL
LIN {X 0,Y 573.628,Z 329.966,A -85,B 0,C 180,E1 -2029.507,E2 -2029.507} C_VEL
LIN {X 0,Y 573.754,Z 318.377,A -85,B 0,C 180,E1 -2029.978,E2 -2029.978} C_VEL
LIN {X 0,Y 573.809,Z 305.475,A -85,B 0,C 180,E1 -2030.354,E2 -2030.354} C_VEL
LIN {X 0,Y 572.939,Z 299.89,A -85,B 0,C 180,E1 -2030.511,E2 -2030.511} C_VEL
LIN {X 0,Y 572.951,Z 296.8,A -85,B 0,C 180,E1 -2033.055,E2 -2033.055} C_VEL
LIN {X 0,Y 572.953,Z 293.684,A -85,B 0,C 180,E1 -2035.65,E2 -2035.65} C_VEL
LIN {X 0,Y 572.942,Z 290.707,A -85,B 0,C 180,E1 -2038.166,E2 -2038.166} C_VEL
LIN {X 0,Y 572.978,Z 287.898,A -85,B 0,C 180,E1 -2040.618,E2 -2040.618} C_VEL
LIN {X 0,Y 573.015,Z 284.788,A -85,B 0,C 180,E1 -2043.552,E2 -2043.552} C_VEL
LIN {X 0,Y 573.049,Z 283.108,A -85,B 0,C 180,E1 -2045.355,E2 -2045.355} C_VEL
LIN {X 0,Y 573.22,Z 283.083,A -85,B 0,C 180,E1 -2047.661,E2 -2047.661} C_VEL
LIN {X 0,Y 573.255,Z 283.078,A -85,B 0,C 180,E1 -2049.923,E2 -2049.923} C_VEL
LIN {X 0,Y 573.261,Z 283.078,A -85,B 0,C 180,E1 -2052.99,E2 -2052.99} C_VEL
LIN {X 0,Y 573.26,Z 283.079,A -85,B 0,C 180,E1 -2055.807,E2 -2055.807} C_VEL
LIN {X 0,Y 573.265,Z 283.081,A -85,B 0,C 180,E1 -2058.745,E2 -2058.745} C_VEL
LIN {X 0,Y 573.287,Z 283.076,A -85,B 0,C 180,E1 -2061.54,E2 -2061.54} C_VEL
LIN {X 0,Y 573.283,Z 283.076,A -85,B 0,C 180,E1 -2064.372,E2 -2064.372} C_VEL
LIN {X 0,Y 573.313,Z 283.074,A -85,B 0,C 180,E1 -2067.892,E2 -2067.892} C_VEL
LIN {X 0,Y 573.332,Z 283.071,A -85,B 0,C 180,E1 -2070.702,E2 -2070.702} C_VEL
LIN {X 0,Y 573.243,Z 283.08,A -85,B 0,C 180,E1 -2073.514,E2 -2073.514} C_VEL
LIN {X 0,Y 573.281,Z 283.077,A -85,B 0,C 180,E1 -2075.628,E2 -2075.628} C_VEL
LIN {X 0,Y 573.284,Z 283.079,A -85,B 0,C 180,E1 -2078.46,E2 -2078.46} C_VEL
LIN {X 0,Y 573.274,Z 283.077,A -85,B 0,C 180,E1 -2081.312,E2 -2081.312} C_VEL
LIN {X 0,Y 573.264,Z 283.077,A -85,B 0,C 180,E1 -2084.417,E2 -2084.417} C_VEL
LIN {X 0,Y 573.256,Z 283.078,A -85,B 0,C 180,E1 -2087.112,E2 -2087.112} C_VEL
LIN {X 0,Y 573.243,Z 283.082,A -85,B 0,C 180,E1 -2090.077,E2 -2090.077} C_VEL
LIN {X 0,Y 573.235,Z 283.081,A -85,B 0,C 180,E1 -2092.338,E2 -2092.338} C_VEL
LIN {X 0,Y 573.25,Z 283.082,A -85,B 0,C 180,E1 -2095.411,E2 -2095.411} C_VEL
LIN {X 0,Y 573.25,Z 283.082,A -85,B 0,C 180,E1 -2098.029,E2 -2098.029} C_VEL
LIN {X 0,Y 573.229,Z 283.083,A -85,B 0,C 180,E1 -2100.993,E2 -2100.993} C_VEL
LIN {X 0,Y 573.243,Z 283.082,A -85,B 0,C 180,E1 -2103.521,E2 -2103.521} C_VEL
LIN {X 0,Y 573.217,Z 283.086,A -85,B 0,C 180,E1 -2106.052,E2 -2106.052} C_VEL
LIN {X 0,Y 573.247,Z 283.082,A -85,B 0,C 180,E1 -2108.702,E2 -2108.702} C_VEL
LIN {X 0,Y 573.23,Z 283.082,A -85,B 0,C 180,E1 -2111.593,E2 -2111.593} C_VEL
LIN {X 0,Y 573.229,Z 283.081,A -85,B 0,C 180,E1 -2114.335,E2 -2114.335} C_VEL
LIN {X 0,Y 573.244,Z 283.08,A -85,B 0,C 180,E1 -2117.359,E2 -2117.359} C_VEL
LIN {X 0,Y 573.25,Z 283.083,A -85,B 0,C 180,E1 -2120.393,E2 -2120.393} C_VEL
LIN {X 0,Y 573.256,Z 283.082,A -85,B 0,C 180,E1 -2123.078,E2 -2123.078} C_VEL
LIN {X 0,Y 573.259,Z 283.082,A -85,B 0,C 180,E1 -2125.671,E2 -2125.671} C_VEL
LIN {X 0,Y 573.241,Z 283.083,A -85,B 0,C 180,E1 -2128.185,E2 -2128.185} C_VEL
LIN {X 0,Y 573.263,Z 283.078,A -85,B 0,C 180,E1 -2130.634,E2 -2130.634} C_VEL
LIN {X 0,Y 573.24,Z 283.084,A -85,B 0,C 180,E1 -2133.508,E2 -2133.508} C_VEL
LIN {X 0,Y 573.219,Z 283.086,A -85,B 0,C 180,E1 -2136.134,E2 -2136.134} C_VEL
LIN {X 0,Y 573.257,Z 283.081,A -85,B 0,C 180,E1 -2138.709,E2 -2138.709} C_VEL
LIN {X 0,Y 573.227,Z 283.086,A -85,B 0,C 180,E1 -2141.411,E2 -2141.411} C_VEL
LIN {X 0,Y 573.241,Z 283.081,A -85,B 0,C 180,E1 -2143.621,E2 -2143.621} C_VEL
LIN {X 0,Y 573.278,Z 283.075,A -85,B 0,C 180,E1 -2145.807,E2 -2145.807} C_VEL
LIN {X 0,Y 573.269,Z 283.076,A -85,B 0,C 180,E1 -2148.745,E2 -2148.745} C_VEL
LIN {X 0,Y 573.257,Z 283.079,A -85,B 0,C 180,E1 -2151.54,E2 -2151.54} C_VEL
LIN {X 0,Y 573.251,Z 283.079,A -85,B 0,C 180,E1 -2153.665,E2 -2153.665} C_VEL
LIN {X 0,Y 573.226,Z 283.085,A -85,B 0,C 180,E1 -2155.781,E2 -2155.781} C_VEL
LIN {X 0,Y 573.318,Z 283.07,A -85,B 0,C 180,E1 -2157.893,E2 -2157.893} C_VEL
LIN {X 0,Y 573.33,Z 283.069,A -85,B 0,C 180,E1 -2160.702,E2 -2160.702} C_VEL
LIN {X 0,Y 573.297,Z 283.074,A -85,B 0,C 180,E1 -2162.811,E2 -2162.811} C_VEL
LIN {X 0,Y 573.293,Z 283.073,A -85,B 0,C 180,E1 -2165.628,E2 -2165.628} C_VEL
LIN {X 0,Y 573.259,Z 283.078,A -85,B 0,C 180,E1 -2168.46,E2 -2168.46} C_VEL
LIN {X 0,Y 573.278,Z 283.077,A -85,B 0,C 180,E1 -2171.312,E2 -2171.312} C_VEL
LIN {X 0,Y 573.274,Z 283.078,A -85,B 0,C 180,E1 -2174.419,E2 -2174.419} C_VEL
LIN {X 0,Y 573.263,Z 283.078,A -85,B 0,C 180,E1 -2177.112,E2 -2177.112} C_VEL
LIN {X 0,Y 573.242,Z 283.08,A -85,B 0,C 180,E1 -2180.077,E2 -2180.077} C_VEL
LIN {X 0,Y 573.235,Z 283.083,A -85,B 0,C 180,E1 -2182.338,E2 -2182.338} C_VEL
LIN {X 0,Y 573.248,Z 283.078,A -85,B 0,C 180,E1 -2185.411,E2 -2185.411} C_VEL
LIN {X 0,Y 573.233,Z 283.084,A -85,B 0,C 180,E1 -2188.565,E2 -2188.565} C_VEL
LIN {X 0,Y 573.223,Z 283.083,A -85,B 0,C 180,E1 -2190.994,E2 -2190.994} C_VEL
LIN {X 0,Y 573.268,Z 283.077,A -85,B 0,C 180,E1 -2193.524,E2 -2193.524} C_VEL
LIN {X 0,Y 573.198,Z 283.086,A -85,B 0,C 180,E1 -2196.053,E2 -2196.053} C_VEL
LIN {X 0,Y 573.241,Z 283.08,A -85,B 0,C 180,E1 -2198.702,E2 -2198.702} C_VEL
LIN {X 0,Y 573.23,Z 283.083,A -85,B 0,C 180,E1 -2201.592,E2 -2201.592} C_VEL
LIN {X 0,Y 573.232,Z 283.084,A -85,B 0,C 180,E1 -2204.334,E2 -2204.334} C_VEL
LIN {X 0,Y 573.237,Z 283.081,A -85,B 0,C 180,E1 -2206.64,E2 -2206.64} C_VEL
LIN {X 0,Y 573.249,Z 283.081,A -85,B 0,C 180,E1 -2209.475,E2 -2209.475} C_VEL
LIN {X 0,Y 573.237,Z 283.085,A -85,B 0,C 180,E1 -2212.192,E2 -2212.192} C_VEL
LIN {X 0,Y 573.288,Z 283.202,A -85,B 0,C 180,E1 -2213.354,E2 -2213.354} C_VEL
LIN {X 0,Y 573.823,Z 288.148,A -85,B 0,C 180,E1 -2214.855,E2 -2214.855} C_VEL
LIN {X 0,Y 573.74,Z 298.104,A -85,B 0,C 180,E1 -2217.695,E2 -2217.695} C_VEL
LIN {X 0,Y 573.568,Z 308.867,A -85,B 0,C 180,E1 -2220.651,E2 -2220.651} C_VEL
LIN {X 0,Y 573.514,Z 319.567,A -85,B 0,C 180,E1 -2223.453,E2 -2223.453} C_VEL
LIN {X 0,Y 573.421,Z 330.079,A -85,B 0,C 180,E1 -2226.143,E2 -2226.143} C_VEL
LIN {X 0,Y 573.327,Z 341.843,A -85,B 0,C 180,E1 -2229.176,E2 -2229.176} C_VEL
LIN {X 0,Y 573.249,Z 352.094,A -85,B 0,C 180,E1 -2231.782,E2 -2231.782} C_VEL
LIN {X 0,Y 573.187,Z 362.345,A -85,B 0,C 180,E1 -2234.351,E2 -2234.351} C_VEL
LIN {X 0,Y 573.113,Z 374.061,A -85,B 0,C 180,E1 -2237.248,E2 -2237.248} C_VEL
LIN {X 0,Y 573.114,Z 374.976,A -85,B 0,C 180,E1 -2237.473,E2 -2237.473} C_VEL
LIN {X 0,Y 573.895,Z 381.224,A -85,B 0,C 180,E1 -2237.603,E2 -2237.603} C_VEL
LIN {X 0,Y 573.791,Z 394.495,A -85,B 0,C 180,E1 -2237.937,E2 -2237.937} C_VEL
LIN {X 0,Y 573.647,Z 407.388,A -85,B 0,C 180,E1 -2238.422,E2 -2238.422} C_VEL
LIN {X 0,Y 573.523,Z 419.954,A -85,B 0,C 180,E1 -2239.061,E2 -2239.061} C_VEL
LIN {X 0,Y 573.453,Z 430.745,A -85,B 0,C 180,E1 -2239.764,E2 -2239.764} C_VEL
LIN {X 0,Y 573.308,Z 439.646,A -85,B 0,C 180,E1 -2240.474,E2 -2240.474} C_VEL
LIN {X 0,Y 573.215,Z 448.786,A -85,B 0,C 180,E1 -2241.362,E2 -2241.362} C_VEL
LIN {X 0,Y 573.142,Z 457.689,A -85,B 0,C 180,E1 -2242.425,E2 -2242.425} C_VEL
LIN {X 0,Y 573.051,Z 464.404,A -85,B 0,C 180,E1 -2243.415,E2 -2243.415} C_VEL
LIN {X 0,Y 573.071,Z 469.68,A -85,B 0,C 180,E1 -2244.37,E2 -2244.37} C_VEL
LIN {X 0,Y 573.028,Z 474.372,A -85,B 0,C 180,E1 -2245.427,E2 -2245.427} C_VEL
LIN {X 0,Y 573.022,Z 477.957,A -85,B 0,C 180,E1 -2246.484,E2 -2246.484} C_VEL
LIN {X 0,Y 572.959,Z 479.808,A -85,B 0,C 180,E1 -2247.188,E2 -2247.188} C_VEL
LIN {X 0,Y 572.94,Z 481.198,A -85,B 0,C 180,E1 -2247.891,E2 -2247.891} C_VEL
LIN {X 0,Y 572.941,Z 482.785,A -85,B 0,C 180,E1 -2249.297,E2 -2249.297} C_VEL
LIN {X 0,Y 572.938,Z 483,A -85,B 0,C 180,E1 -2250,E2 -2250} C_VEL
LIN {X 0,Y 572.946,Z 482.186,A -85,B 0,C 180,E1 -2251.406,E2 -2251.406} C_VEL
LIN {X 0,Y 572.94,Z 481.2,A -85,B 0,C 180,E1 -2252.109,E2 -2252.109} C_VEL
LIN {X 0,Y 572.959,Z 479.81,A -85,B 0,C 180,E1 -2252.812,E2 -2252.812} C_VEL
LIN {X 0,Y 573.015,Z 476.896,A -85,B 0,C 180,E1 -2253.868,E2 -2253.868} C_VEL
LIN {X 0,Y 572.963,Z 472.949,A -85,B 0,C 180,E1 -2254.926,E2 -2254.926} C_VEL
LIN {X 0,Y 573.065,Z 466.876,A -85,B 0,C 180,E1 -2256.16,E2 -2256.16} C_VEL
LIN {X 0,Y 573.119,Z 460.237,A -85,B 0,C 180,E1 -2257.221,E2 -2257.221} C_VEL
LIN {X 0,Y 573.201,Z 451.99,A -85,B 0,C 180,E1 -2258.283,E2 -2258.283} C_VEL
LIN {X 0,Y 573.287,Z 443.537,A -85,B 0,C 180,E1 -2259.17,E2 -2259.17} C_VEL
LIN {X 0,Y 573.427,Z 433.096,A -85,B 0,C 180,E1 -2260.058,E2 -2260.058} C_VEL
LIN {X 0,Y 573.524,Z 421.523,A -85,B 0,C 180,E1 -2260.848,E2 -2260.848} C_VEL
LIN {X 0,Y 573.614,Z 409.881,A -85,B 0,C 180,E1 -2261.466,E2 -2261.466} C_VEL
LIN {X 0,Y 573.751,Z 397.169,A -85,B 0,C 180,E1 -2261.974,E2 -2261.974} C_VEL
LIN {X 0,Y 573.849,Z 384.514,A -85,B 0,C 180,E1 -2262.331,E2 -2262.331} C_VEL
LIN {X 0,Y 573.617,Z 378.153,A -85,B 0,C 180,E1 -2262.463,E2 -2262.463} C_VEL
LIN {X 0,Y 573.115,Z 374.976,A -85,B 0,C 180,E1 -2262.527,E2 -2262.527} C_VEL
LIN {X 0,Y 573.18,Z 363.81,A -85,B 0,C 180,E1 -2265.285,E2 -2265.285} C_VEL
LIN {X 0,Y 573.253,Z 353.558,A -85,B 0,C 180,E1 -2267.848,E2 -2267.848} C_VEL
LIN {X 0,Y 573.31,Z 343.307,A -85,B 0,C 180,E1 -2270.449,E2 -2270.449} C_VEL
LIN {X 0,Y 573.386,Z 332.727,A -85,B 0,C 180,E1 -2273.179,E2 -2273.179} C_VEL
LIN {X 0,Y 573.473,Z 320.791,A -85,B 0,C 180,E1 -2276.18,E2 -2276.18} C_VEL
LIN {X 0,Y 573.477,Z 309.907,A -85,B 0,C 180,E1 -2278.952,E2 -2278.952} C_VEL
LIN {X 0,Y 573.574,Z 299.424,A -85,B 0,C 180,E1 -2281.795,E2 -2281.795} C_VEL
LIN {X 0,Y 573.71,Z 290.502,A -85,B 0,C 180,E1 -2284.299,E2 -2284.299} C_VEL
LIN {X 0,Y 573.714,Z 286.131,A -85,B 0,C 180,E1 -2285.583,E2 -2285.583} C_VEL
LIN {X 0,Y 573.244,Z 283.083,A -85,B 0,C 180,E1 -2286.595,E2 -2286.595} C_VEL
LIN {X 0,Y 573.245,Z 283.081,A -85,B 0,C 180,E1 -2289.608,E2 -2289.608} C_VEL
LIN {X 0,Y 573.244,Z 283.082,A -85,B 0,C 180,E1 -2292.642,E2 -2292.642} C_VEL
LIN {X 0,Y 573.241,Z 283.083,A -85,B 0,C 180,E1 -2295.667,E2 -2295.667} C_VEL
LIN {X 0,Y 573.234,Z 283.083,A -85,B 0,C 180,E1 -2298.543,E2 -2298.543} C_VEL
LIN {X 0,Y 573.254,Z 283.081,A -85,B 0,C 180,E1 -2301.299,E2 -2301.299} C_VEL
LIN {X 0,Y 573.218,Z 283.087,A -85,B 0,C 180,E1 -2304.018,E2 -2304.018} C_VEL
LIN {X 0,Y 573.275,Z 283.077,A -85,B 0,C 180,E1 -2306.518,E2 -2306.518} C_VEL
LIN {X 0,Y 573.244,Z 283.083,A -85,B 0,C 180,E1 -2309.116,E2 -2309.116} C_VEL
LIN {X 0,Y 573.256,Z 283.081,A -85,B 0,C 180,E1 -2311.971,E2 -2311.971} C_VEL
LIN {X 0,Y 573.261,Z 283.079,A -85,B 0,C 180,E1 -2314.59,E2 -2314.59} C_VEL
LIN {X 0,Y 573.241,Z 283.081,A -85,B 0,C 180,E1 -2317.662,E2 -2317.662} C_VEL
LIN {X 0,Y 573.272,Z 283.078,A -85,B 0,C 180,E1 -2320.67,E2 -2320.67} C_VEL
LIN {X 0,Y 573.248,Z 283.081,A -85,B 0,C 180,E1 -2323.622,E2 -2323.622} C_VEL
LIN {X 0,Y 573.28,Z 283.077,A -85,B 0,C 180,E1 -2325.807,E2 -2325.807} C_VEL
LIN {X 0,Y 573.27,Z 283.078,A -85,B 0,C 180,E1 -2328.745,E2 -2328.745} C_VEL
LIN {X 0,Y 573.26,Z 283.079,A -85,B 0,C 180,E1 -2331.54,E2 -2331.54} C_VEL
LIN {X 0,Y 573.29,Z 283.076,A -85,B 0,C 180,E1 -2334.372,E2 -2334.372} C_VEL
LIN {X 0,Y 573.318,Z 283.073,A -85,B 0,C 180,E1 -2337.892,E2 -2337.892} C_VEL
LIN {X 0,Y 573.333,Z 283.07,A -85,B 0,C 180,E1 -2340.702,E2 -2340.702} C_VEL
LIN {X 0,Y 573.307,Z 283.074,A -85,B 0,C 180,E1 -2342.811,E2 -2342.811} C_VEL
LIN {X 0,Y 573.295,Z 283.075,A -85,B 0,C 180,E1 -2345.628,E2 -2345.628} C_VEL
LIN {X 0,Y 573.263,Z 283.08,A -85,B 0,C 180,E1 -2348.46,E2 -2348.46} C_VEL
LIN {X 0,Y 573.05,Z 283.216,A -85,B 0,C 180,E1 -2350.601,E2 -2350.601} C_VEL
LIN {X 0,Y 573.049,Z 285.345,A -85,B 0,C 180,E1 -2352.753,E2 -2352.753} C_VEL
LIN {X 0,Y 573.027,Z 287.378,A -85,B 0,C 180,E1 -2354.925,E2 -2354.925} C_VEL
LIN {X 0,Y 572.94,Z 290.629,A -85,B 0,C 180,E1 -2357.858,E2 -2357.858} C_VEL
LIN {X 0,Y 572.965,Z 293.263,A -85,B 0,C 180,E1 -2360.087,E2 -2360.087} C_VEL
LIN {X 0,Y 572.939,Z 296.893,A -85,B 0,C 180,E1 -2363.112,E2 -2363.112} C_VEL
